C07161=1019.508,345.126,-145.599,171.167,50.075,159.868
C07162=1019.516,345.374,-145.635,171.174,50.072,159.868
C07163=1019.523,345.620,-145.671,171.182,50.070,159.869
C07164=1019.530,345.867,-145.708,171.189,50.068,159.869
C07165=1019.538,346.115,-145.744,171.196,50.066,159.870
C07166=1019.545,346.362,-145.781,171.203,50.064,159.871
C07167=1019.553,346.609,-145.818,171.210,50.062,159.872
C07168=1019.560,346.857,-145.854,171.217,50.060,159.872
C07169=1019.568,347.104,-145.891,171.225,50.058,159.873
C07170=1019.575,347.352,-145.928,171.232,50.055,159.874
C07171=1019.582,347.598,-145.965,171.239,50.054,159.874
C07172=1019.590,347.845,-146.002,171.247,50.052,159.875
C07173=1019.597,348.093,-146.039,171.254,50.050,159.876
C07174=1019.605,348.339,-146.076,171.261,50.048,159.877
C07175=1019.612,348.586,-146.113,171.269,50.046,159.877
C07176=1019.620,348.834,-146.150,171.277,50.044,159.878
C07177=1019.627,349.081,-146.187,171.284,50.042,159.879
C07178=1019.635,349.328,-146.224,171.291,50.040,159.880
C07179=1019.642,349.575,-146.262,171.299,50.038,159.880
C07180=1019.649,349.823,-146.298,171.306,50.036,159.881
C07181=1019.657,350.070,-146.335,171.314,50.034,159.882
C07182=1019.664,350.317,-146.373,171.321,50.033,159.883
C07183=1019.672,350.564,-146.410,171.328,50.031,159.884
C07184=1019.680,350.811,-146.447,171.336,50.029,159.884
C07185=1019.687,351.058,-146.485,171.343,50.027,159.885
C07186=1019.695,351.305,-146.522,171.351,50.025,159.886
C07187=1019.703,351.552,-146.560,171.358,50.023,159.887
C07188=1019.710,351.799,-146.596,171.366,50.021,159.887
C07189=1019.717,352.046,-146.634,171.374,50.020,159.888
C07190=1019.725,352.293,-146.671,171.381,50.018,159.889
C07191=1019.733,352.539,-146.709,171.388,50.016,159.890
C07192=1019.741,352.786,-146.746,171.396,50.015,159.891
C07193=1019.748,353.033,-146.783,171.404,50.013,159.892
C07194=1019.756,353.280,-146.820,171.412,50.011,159.892
C07195=1019.764,353.526,-146.859,171.419,50.009,159.893
C07196=1019.772,353.773,-146.896,171.426,50.007,159.894
C07197=1019.779,354.020,-146.933,171.434,50.005,159.895
C07198=1019.787,354.268,-146.971,171.443,50.004,159.896
C07199=1019.795,354.514,-147.009,171.450,50.002,159.897
C07200=1019.802,354.761,-147.046,171.457,50.000,159.897
C07201=1019.810,355.008,-147.084,171.465,49.999,159.898
C07202=1019.818,355.256,-147.122,171.473,49.998,159.899
C07203=1019.825,355.503,-147.160,171.480,49.996,159.900
C07204=1019.833,355.749,-147.197,171.489,49.994,159.901
C07205=1019.841,355.997,-147.235,171.496,49.993,159.902
C07206=1019.848,356.244,-147.274,171.503,49.991,159.903
C07207=1019.856,356.491,-147.311,171.511,49.990,159.904
C07208=1019.864,356.738,-147.350,171.520,49.987,159.905
C07209=1019.872,356.984,-147.387,171.527,49.986,159.906
C07210=1019.880,357.232,-147.425,171.535,49.985,159.906
C07211=1019.888,357.478,-147.463,171.543,49.983,159.907
C07212=1019.895,357.726,-147.501,171.551,49.981,159.908
C07213=1019.903,357.973,-147.540,171.559,49.980,159.909
C07214=1019.910,358.219,-147.578,171.567,49.979,159.910
C07215=1019.919,358.466,-147.616,171.575,49.977,159.911
C07216=1019.927,358.713,-147.653,171.583,49.976,159.912
C07217=1019.935,358.961,-147.692,171.590,49.975,159.913
C07218=1019.942,359.207,-147.730,171.598,49.973,159.914
C07219=1019.950,359.454,-147.769,171.607,49.971,159.915
C07220=1019.958,359.701,-147.807,171.614,49.970,159.916
C07221=1019.966,359.948,-147.846,171.622,49.969,159.917
C07222=1019.974,360.195,-147.884,171.631,49.967,159.918
C07223=1019.982,360.442,-147.923,171.638,49.966,159.919
C07224=1019.989,360.688,-147.961,171.646,49.965,159.920
C07225=1019.997,360.936,-148.000,171.655,49.963,159.921
C07226=1020.005,361.183,-148.039,171.663,49.962,159.922
C07227=1020.013,361.430,-148.077,171.670,49.961,159.923
C07228=1020.021,361.676,-148.116,171.678,49.960,159.924
C07229=1020.029,361.923,-148.154,171.687,49.958,159.925
C07230=1020.037,362.170,-148.193,171.695,49.957,159.926
C07231=1020.045,362.417,-148.232,171.703,49.955,159.927
C07232=1020.053,362.663,-148.271,171.711,49.954,159.928
C07233=1020.060,362.910,-148.310,171.719,49.953,159.929
C07234=1020.068,363.158,-148.348,171.728,49.952,159.930
C07235=1020.077,363.404,-148.388,171.735,49.951,159.931
C07236=1020.084,363.651,-148.426,171.743,49.949,159.932
C07237=1020.092,363.898,-148.465,171.752,49.948,159.933
C07238=1020.101,364.145,-148.504,171.760,49.947,159.934
C07239=1020.109,364.392,-148.543,171.769,49.946,159.935
C07240=1020.117,364.638,-148.581,171.777,49.945,159.936
C07241=1020.124,364.885,-148.621,171.785,49.943,159.937
C07242=1020.133,365.132,-148.660,171.794,49.943,159.939
C07243=1020.141,365.379,-148.699,171.802,49.941,159.940
C07244=1020.149,365.626,-148.738,171.810,49.940,159.941
C07245=1020.158,365.872,-148.777,171.818,49.939,159.942
C07246=1020.166,366.119,-148.816,171.827,49.938,159.943
C07247=1020.174,366.366,-148.855,171.835,49.937,159.944
C07248=1020.182,366.620,-148.895,171.844,49.936,159.945
C07249=1020.191,366.874,-148.936,171.853,49.934,159.946
C07250=1020.199,367.127,-148.977,171.862,49.933,159.947
C07251=1020.208,367.381,-149.017,171.870,49.932,159.948
C07252=1020.216,367.628,-149.056,171.879,49.931,159.950
C07253=1020.225,367.875,-149.095,171.887,49.930,159.951
C07254=1020.232,368.122,-149.135,171.896,49.929,159.952
C07255=1020.241,368.369,-149.174,171.904,49.929,159.953
C07256=1020.249,368.615,-149.213,171.913,49.927,159.954
C07257=1020.257,368.861,-149.254,171.922,49.926,159.956
C07258=1020.266,369.108,-149.293,171.930,49.926,159.957
C07259=1020.273,369.355,-149.333,171.939,49.925,159.958
C07260=1020.282,369.602,-149.373,171.947,49.924,159.959
C07261=1020.290,369.848,-149.413,171.956,49.923,159.960
C07262=1020.298,370.095,-149.452,171.964,49.922,159.961
C07263=1020.306,370.341,-149.493,171.973,49.921,159.963
C07264=1020.315,370.588,-149.532,171.981,49.921,159.964
C07265=1020.322,370.835,-149.572,171.990,49.920,159.965
C07266=1020.332,371.082,-149.612,171.999,49.918,159.966
C07267=1020.339,371.328,-149.652,172.007,49.918,159.967
C07268=1020.348,371.575,-149.691,172.017,49.917,159.969
C07269=1020.356,371.821,-149.732,172.026,49.916,159.970
C07270=1020.364,372.068,-149.771,172.034,49.916,159.971
C07271=1020.374,372.315,-149.812,172.043,49.915,159.973
C07272=1020.381,372.562,-149.852,172.052,49.914,159.974
C07273=1020.390,372.807,-149.892,172.060,49.913,159.975
C07274=1020.398,373.054,-149.932,172.070,49.913,159.976
C07275=1020.407,373.301,-149.972,172.079,49.912,159.978
C07276=1020.415,373.548,-150.012,172.087,49.911,159.979
C07277=1020.424,373.794,-150.052,172.096,49.911,159.980
C07278=1020.432,374.041,-150.093,172.105,49.910,159.981
C07279=1020.441,374.288,-150.132,172.113,49.909,159.983
C07280=1020.449,374.535,-150.173,172.123,49.909,159.984
C07281=1020.458,374.780,-150.213,172.132,49.908,159.985
C07282=1020.466,375.027,-150.254,172.141,49.907,159.987
C07283=1020.475,375.274,-150.294,172.150,49.907,159.988
C07284=1020.483,375.520,-150.334,172.159,49.906,159.989
C07285=1020.493,375.767,-150.375,172.168,49.905,159.991
C07286=1020.501,376.013,-150.415,172.178,49.905,159.992
C07287=1020.510,376.260,-150.456,172.187,49.904,159.993
C07288=1020.518,376.506,-150.496,172.195,49.904,159.995
C07289=1020.527,376.753,-150.537,172.204,49.903,159.996
C07290=1020.535,377.000,-150.578,172.214,49.903,159.998
C07291=1020.544,377.246,-150.619,172.223,49.902,159.999
C07292=1020.552,377.492,-150.660,172.232,49.902,160.000
C07293=1020.561,377.739,-150.701,172.241,49.902,160.002
C07294=1020.569,377.985,-150.741,172.250,49.901,160.003
C07295=1020.578,378.232,-150.782,172.260,49.900,160.005
C07296=1020.587,378.478,-150.824,172.269,49.900,160.006
C07297=1020.595,378.724,-150.864,172.279,49.900,160.007
C07298=1020.604,378.971,-150.906,172.288,49.899,160.009
C07299=1020.613,379.218,-150.947,172.297,49.899,160.010
C07300=1020.621,379.464,-150.988,172.306,49.899,160.012
C07301=1020.630,379.710,-151.029,172.315,49.898,160.013
C07302=1020.639,379.957,-151.070,172.325,49.898,160.015
C07303=1020.648,380.203,-151.111,172.334,49.898,160.016
C07304=1020.657,380.449,-151.153,172.344,49.897,160.018
C07305=1020.665,380.696,-151.194,172.353,49.897,160.019
C07306=1020.674,380.943,-151.236,172.363,49.897,160.021
C07307=1020.683,381.190,-151.277,172.372,49.896,160.022
C07308=1020.693,381.465,-151.322,172.383,49.896,160.024
C07309=1020.703,381.741,-151.368,172.394,49.896,160.025
C07310=1020.712,382.017,-151.415,172.405,49.896,160.027
C07311=1020.723,382.292,-151.462,172.415,49.895,160.029
C07312=1020.731,382.539,-151.503,172.425,49.895,160.030
C07313=1020.740,382.786,-151.545,172.435,49.895,160.032
C07314=1020.750,383.032,-151.586,172.444,49.895,160.033
C07315=1020.759,383.278,-151.628,172.454,49.894,160.035
C07316=1020.768,383.525,-151.669,172.463,49.894,160.036
C07317=1020.777,383.771,-151.711,172.473,49.894,160.038
C07318=1020.786,384.017,-151.753,172.483,49.894,160.040
C07319=1020.795,384.263,-151.794,172.492,49.893,160.041
C07320=1020.804,384.510,-151.836,172.503,49.893,160.043
C07321=1020.813,384.756,-151.877,172.513,49.893,160.044
C07322=1020.822,385.002,-151.919,172.522,49.893,160.046
C07323=1020.831,385.249,-151.961,172.532,49.893,160.047
C07324=1020.840,385.495,-152.003,172.542,49.893,160.049
C07325=1020.849,385.741,-152.045,172.551,49.893,160.051
C07326=1020.859,385.988,-152.087,172.562,49.893,160.052
C07327=1020.868,386.234,-152.129,172.572,49.893,160.054
C07328=1020.877,386.480,-152.171,172.582,49.893,160.056
C07329=1020.886,386.726,-152.214,172.592,49.893,160.057
C07330=1020.895,386.972,-152.255,172.601,49.893,160.059
C07331=1020.904,387.218,-152.298,172.612,49.893,160.060
C07332=1020.914,387.465,-152.340,172.622,49.893,160.062
C07333=1020.923,387.711,-152.382,172.632,49.893,160.064
C07334=1020.932,387.957,-152.424,172.642,49.893,160.066
C07335=1020.941,388.203,-152.466,172.652,49.893,160.067
C07336=1020.951,388.449,-152.509,172.662,49.894,160.069
C07337=1020.959,388.696,-152.551,172.672,49.894,160.071
C07338=1020.969,388.942,-152.594,172.682,49.894,160.072
C07339=1020.978,389.188,-152.637,172.693,49.894,160.074
C07340=1020.988,389.434,-152.679,172.703,49.894,160.076
C07341=1020.996,389.680,-152.722,172.713,49.894,160.078
C07342=1021.006,389.926,-152.765,172.724,49.894,160.079
C07343=1021.015,390.172,-152.807,172.734,49.895,160.081
C07344=1021.025,390.419,-152.850,172.744,49.895,160.083
C07345=1021.034,390.664,-152.893,172.754,49.895,160.084
C07346=1021.043,390.911,-152.936,172.765,49.896,160.086
C07347=1021.053,391.157,-152.978,172.776,49.895,160.088
C07348=1021.063,391.403,-153.021,172.785,49.896,160.090
C07349=1021.072,391.648,-153.064,172.796,49.897,160.092
C07350=1021.081,391.895,-153.108,172.807,49.896,160.094
C07351=1021.090,392.141,-153.150,172.816,49.897,160.095
C07352=1021.100,392.387,-153.193,172.828,49.897,160.097
C07353=1021.110,392.632,-153.236,172.838,49.897,160.099
C07354=1021.119,392.879,-153.280,172.849,49.898,160.101
C07355=1021.129,393.126,-153.322,172.859,49.898,160.103
C07356=1021.138,393.371,-153.366,172.870,49.899,160.105
C07357=1021.147,393.618,-153.409,172.880,49.899,160.106
C07358=1021.158,393.863,-153.452,172.891,49.899,160.108
C07359=1021.166,394.109,-153.496,172.902,49.900,160.110
C07360=1021.176,394.355,-153.539,172.913,49.901,160.112
C07361=1021.186,394.601,-153.583,172.923,49.901,160.114
C07362=1021.195,394.846,-153.626,172.934,49.901,160.116
C07363=1021.205,395.093,-153.669,172.945,49.902,160.118
C07364=1021.214,395.339,-153.713,172.955,49.903,160.120
C07365=1021.225,395.585,-153.757,172.967,49.903,160.122
C07366=1021.234,395.831,-153.801,172.977,49.904,160.124
C07367=1021.244,396.076,-153.844,172.988,49.904,160.125
C07368=1021.256,396.390,-153.900,173.002,49.905,160.128
C07369=1021.268,396.703,-153.955,173.016,49.906,160.131
C07370=1021.281,397.017,-154.011,173.030,49.906,160.133
C07371=1021.294,397.330,-154.066,173.044,49.907,160.135
C07372=1021.303,397.576,-154.110,173.055,49.907,160.137
C07373=1021.313,397.822,-154.155,173.067,49.908,160.140
C07374=1021.323,398.067,-154.199,173.078,49.909,160.142
C07375=1021.333,398.313,-154.243,173.088,49.910,160.143
C07376=1021.343,398.559,-154.286,173.099,49.910,160.145
C07377=1021.352,398.805,-154.331,173.111,49.911,160.148
C07378=1021.363,399.051,-154.375,173.122,49.912,160.150
C07379=1021.372,399.297,-154.419,173.134,49.913,160.152
C07380=1021.382,399.542,-154.464,173.144,49.913,160.154
C07381=1021.392,399.788,-154.507,173.155,49.914,160.156
C07382=1021.402,400.034,-154.552,173.167,49.915,160.158
C07383=1021.412,400.280,-154.597,173.179,49.916,160.160
C07384=1021.422,400.526,-154.641,173.190,49.916,160.162
C07385=1021.432,400.771,-154.686,173.202,49.917,160.164
C07386=1021.441,401.017,-154.730,173.213,49.918,160.166
C07387=1021.452,401.263,-154.774,173.225,49.919,160.169
C07388=1021.462,401.509,-154.819,173.236,49.920,160.171
C07389=1021.472,401.754,-154.864,173.248,49.921,160.173
C07390=1021.481,402.000,-154.909,173.259,49.922,160.175
C07391=1021.492,402.246,-154.954,173.271,49.922,160.177
C07392=1021.501,402.491,-154.999,173.282,49.923,160.179
C07393=1021.512,402.737,-155.043,173.294,49.924,160.181
C07394=1021.522,402.983,-155.088,173.306,49.925,160.184
C07395=1021.532,403.228,-155.133,173.317,49.926,160.186
C07396=1021.542,403.475,-155.178,173.329,49.927,160.188
C07397=1021.552,403.720,-155.223,173.341,49.928,160.190
C07398=1021.563,403.965,-155.268,173.352,49.929,160.192
C07399=1021.573,404.211,-155.313,173.364,49.931,160.195
C07400=1021.583,404.456,-155.358,173.376,49.932,160.197
C07401=1021.593,404.702,-155.404,173.388,49.933,160.199
C07402=1021.604,404.948,-155.449,173.399,49.934,160.202
C07403=1021.613,405.194,-155.494,173.412,49.935,160.204
C07404=1021.625,405.439,-155.539,173.424,49.936,160.206
C07405=1021.634,405.684,-155.584,173.436,49.937,160.208
C07406=1021.645,405.930,-155.630,173.448,49.939,160.211
C07407=1021.655,406.176,-155.675,173.460,49.939,160.213
C07408=1021.666,406.422,-155.721,173.472,49.941,160.216
C07409=1021.677,406.666,-155.766,173.484,49.942,160.218
C07410=1021.687,406.913,-155.811,173.496,49.943,160.220
C07411=1021.698,407.158,-155.857,173.509,49.944,160.222
C07412=1021.708,407.404,-155.903,173.521,49.945,160.225
C07413=1021.719,407.650,-155.948,173.533,49.946,160.227
C07414=1021.729,407.895,-155.994,173.545,49.948,160.230
C07415=1021.740,408.140,-156.039,173.557,49.949,160.232
C07416=1021.751,408.386,-156.085,173.570,49.950,160.234
C07417=1021.761,408.631,-156.131,173.582,49.951,160.237
C07418=1021.772,408.877,-156.177,173.595,49.952,160.239
C07419=1021.782,409.123,-156.223,173.607,49.954,160.242
C07420=1021.793,409.368,-156.269,173.620,49.955,160.244
C07421=1021.804,409.614,-156.314,173.632,49.957,160.246
C07422=1021.815,409.859,-156.361,173.645,49.958,160.249
C07423=1021.825,410.104,-156.407,173.657,49.959,160.251
C07424=1021.836,410.350,-156.453,173.671,49.961,160.254
C07425=1021.846,410.595,-156.500,173.683,49.963,160.256
C07426=1021.857,410.841,-156.546,173.696,49.964,160.259
C07427=1021.868,411.086,-156.593,173.708,49.965,160.261
C07428=1021.881,411.399,-156.652,173.724,49.968,160.265
C07429=1021.895,411.712,-156.711,173.741,49.969,160.268
C07430=1021.910,412.026,-156.770,173.757,49.971,160.271
C07431=1021.923,412.338,-156.829,173.773,49.973,160.274
C07432=1021.934,412.584,-156.876,173.786,49.975,160.277
C07433=1021.945,412.829,-156.923,173.799,49.976,160.280
C07434=1021.956,413.074,-156.969,173.813,49.978,160.282
C07435=1021.967,413.320,-157.016,173.825,49.979,160.285
C07436=1021.978,413.565,-157.063,173.838,49.981,160.287
C07437=1021.989,413.810,-157.110,173.852,49.983,160.290
C07438=1022.000,414.055,-157.157,173.865,49.984,160.293
C07439=1022.011,414.300,-157.203,173.878,49.986,160.295
C07440=1022.022,414.546,-157.251,173.892,49.987,160.298
C07441=1022.033,414.791,-157.298,173.904,49.989,160.301
C07442=1022.045,415.037,-157.345,173.917,49.991,160.303
C07443=1022.056,415.283,-157.392,173.931,49.993,160.306
C07444=1022.067,415.528,-157.438,173.944,49.994,160.309
C07445=1022.078,415.773,-157.486,173.958,49.996,160.312
C07446=1022.089,416.018,-157.533,173.971,49.998,160.314
C07447=1022.100,416.263,-157.581,173.985,49.999,160.317
C07448=1022.112,416.509,-157.628,173.998,50.002,160.320
C07449=1022.122,416.754,-157.676,174.012,50.003,160.323
C07450=1022.134,416.999,-157.723,174.025,50.005,160.325
C07451=1022.146,417.244,-157.771,174.039,50.007,160.328
C07452=1022.156,417.489,-157.819,174.052,50.009,160.331
C07453=1022.168,417.735,-157.866,174.067,50.011,160.334
C07454=1022.179,417.980,-157.914,174.081,50.013,160.337
C07455=1022.191,418.225,-157.962,174.094,50.015,160.340
C07456=1022.202,418.470,-158.010,174.108,50.016,160.342
C07457=1022.213,418.716,-158.058,174.122,50.019,160.345
C07458=1022.225,418.960,-158.105,174.136,50.021,160.348
C07459=1022.236,419.205,-158.154,174.150,50.022,160.351
C07460=1022.248,419.450,-158.201,174.164,50.024,160.354
C07461=1022.259,419.695,-158.249,174.177,50.027,160.357
C07462=1022.271,419.941,-158.297,174.192,50.028,160.360
C07463=1022.282,420.186,-158.345,174.206,50.031,160.363
C07464=1022.294,420.432,-158.394,174.221,50.033,160.366
C07465=1022.306,420.676,-158.442,174.235,50.035,160.369
C07466=1022.318,420.921,-158.490,174.249,50.037,160.372
C07467=1022.329,421.167,-158.538,174.263,50.039,160.375
C07468=1022.341,421.411,-158.586,174.277,50.041,160.378
C07469=1022.352,421.657,-158.635,174.292,50.043,160.381
C07470=1022.365,421.902,-158.684,174.306,50.045,160.384
C07471=1022.376,422.147,-158.732,174.321,50.047,160.387
C07472=1022.389,422.415,-158.785,174.336,50.050,160.390
C07473=1022.402,422.683,-158.839,174.352,50.052,160.393
C07474=1022.415,422.951,-158.892,174.369,50.054,160.397
C07475=1022.428,423.219,-158.945,174.384,50.057,160.400
C07476=1022.439,423.463,-158.994,174.399,50.059,160.403
C07477=1022.451,423.709,-159.043,174.414,50.062,160.407
C07478=1022.464,423.953,-159.092,174.428,50.064,160.410
C07479=1022.476,424.199,-159.141,174.443,50.066,160.413
C07480=1022.488,424.443,-159.190,174.459,50.068,160.416
C07481=1022.500,424.689,-159.239,174.474,50.071,160.419
C07482=1022.511,424.933,-159.288,174.488,50.073,160.422
C07483=1022.524,425.178,-159.338,174.503,50.076,160.426
C07484=1022.536,425.423,-159.387,174.518,50.078,160.429
C07485=1022.548,425.668,-159.436,174.534,50.080,160.432
C07486=1022.560,425.913,-159.486,174.549,50.083,160.435
C07487=1022.572,426.157,-159.534,174.564,50.085,160.439
C07488=1022.588,426.479,-159.600,174.584,50.089,160.443
C07489=1022.604,426.800,-159.665,174.604,50.091,160.447
C07490=1022.620,427.120,-159.731,174.624,50.095,160.452
C07491=1022.636,427.441,-159.796,174.644,50.098,160.456
C07492=1022.648,427.685,-159.845,174.660,50.101,160.459
C07493=1022.661,427.930,-159.895,174.675,50.103,160.463
C07494=1022.673,428.175,-159.945,174.691,50.106,160.466
C07495=1022.685,428.420,-159.996,174.706,50.109,160.470
C07496=1022.697,428.665,-160.046,174.722,50.111,160.473
C07497=1022.710,428.909,-160.096,174.738,50.114,160.476
C07498=1022.723,429.154,-160.145,174.754,50.116,160.480
C07499=1022.735,429.399,-160.195,174.769,50.119,160.483
C07500=1022.747,429.643,-160.245,174.785,50.122,160.487
C07501=1022.760,429.888,-160.296,174.802,50.125,160.490
C07502=1022.772,430.133,-160.346,174.817,50.127,160.494
C07503=1022.785,430.377,-160.396,174.834,50.130,160.497
C07504=1022.799,430.622,-160.447,174.849,50.133,160.501
C07505=1022.811,430.867,-160.497,174.866,50.135,160.504
C07506=1022.824,431.111,-160.548,174.881,50.138,160.508
C07507=1022.836,431.355,-160.599,174.898,50.141,160.511
C07508=1022.849,431.601,-160.649,174.914,50.144,160.515
C07509=1022.862,431.845,-160.700,174.931,50.147,160.519
C07510=1022.875,432.089,-160.750,174.947,50.149,160.522
C07511=1022.888,432.334,-160.801,174.964,50.152,160.526
C07512=1022.901,432.578,-160.851,174.980,50.155,160.529
C07513=1022.914,432.823,-160.903,174.997,50.158,160.533
C07514=1022.927,433.067,-160.954,175.013,50.161,160.537
C07515=1022.939,433.311,-161.005,175.030,50.164,160.540
C07516=1022.953,433.556,-161.056,175.047,50.166,160.544
C07517=1022.965,433.800,-161.107,175.064,50.169,160.548
C07518=1022.978,434.045,-161.158,175.081,50.172,160.552
C07519=1022.992,434.289,-161.210,175.097,50.176,160.555
C07520=1023.005,434.534,-161.261,175.114,50.179,160.559
C07521=1023.018,434.778,-161.313,175.131,50.182,160.563
C07522=1023.031,435.023,-161.365,175.148,50.185,160.567
C07523=1023.044,435.267,-161.416,175.165,50.188,160.571
C07524=1023.057,435.512,-161.467,175.182,50.191,160.574
C07525=1023.070,435.756,-161.519,175.199,50.194,160.578
C07526=1023.084,436.000,-161.571,175.217,50.197,160.582
C07527=1023.097,436.244,-161.623,175.235,50.200,160.586
C07528=1023.110,436.488,-161.674,175.252,50.203,160.590
C07529=1023.124,436.732,-161.726,175.269,50.207,160.594
C07530=1023.137,436.977,-161.778,175.286,50.210,160.598
C07531=1023.150,437.221,-161.831,175.304,50.212,160.602
C07532=1023.164,437.465,-161.883,175.322,50.216,160.606
C07533=1023.177,437.710,-161.934,175.339,50.219,160.610
C07534=1023.191,437.954,-161.986,175.357,50.222,160.614
C07535=1023.204,438.198,-162.039,175.375,50.226,160.618
C07536=1022.814,436.266,-161.961,175.226,50.266,160.605
C07537=1022.801,436.022,-161.909,175.209,50.264,160.601
C07538=1022.788,435.777,-161.858,175.191,50.260,160.597
C07539=1022.774,435.533,-161.806,175.174,50.257,160.593
C07540=1022.761,435.289,-161.754,175.157,50.254,160.589
C07541=1022.748,435.044,-161.703,175.139,50.252,160.585
C07542=1022.735,434.800,-161.651,175.122,50.248,160.581
C07543=1022.722,434.556,-161.600,175.105,50.245,160.578
C07544=1022.708,434.312,-161.549,175.088,50.243,160.574
C07545=1022.695,434.067,-161.497,175.071,50.240,160.570
C07546=1022.683,433.823,-161.447,175.054,50.237,160.567
C07547=1022.669,433.578,-161.395,175.038,50.234,160.563
C07548=1022.656,433.334,-161.344,175.021,50.231,160.559
C07549=1022.643,433.089,-161.293,175.004,50.228,160.555
C07550=1022.631,432.845,-161.242,174.988,50.226,160.552
C07551=1022.618,432.601,-161.191,174.971,50.223,160.548
C07552=1022.605,432.356,-161.140,174.955,50.220,160.544
C07553=1022.592,432.112,-161.089,174.938,50.217,160.541
C07554=1022.579,431.867,-161.038,174.922,50.215,160.537
C07555=1022.567,431.622,-160.988,174.905,50.212,160.534
C07556=1022.554,431.378,-160.937,174.889,50.209,160.530
C07557=1022.540,431.133,-160.886,174.873,50.206,160.526
C07558=1022.528,430.888,-160.836,174.857,50.204,160.523
C07559=1022.515,430.644,-160.786,174.840,50.201,160.519
C07560=1022.503,430.399,-160.735,174.825,50.198,160.516
C07561=1022.490,430.154,-160.685,174.808,50.196,160.512
C07562=1022.477,429.911,-160.635,174.792,50.193,160.509
C07563=1022.464,429.665,-160.585,174.776,50.191,160.505
C07564=1022.452,429.420,-160.535,174.760,50.188,160.502
C07565=1022.439,429.176,-160.484,174.744,50.186,160.499
C07566=1022.427,428.931,-160.434,174.729,50.183,160.495
C07567=1022.415,428.686,-160.384,174.713,50.180,160.492
C07568=1022.402,428.442,-160.334,174.697,50.178,160.488
C07569=1022.390,428.198,-160.284,174.681,50.176,160.485
C07570=1022.378,427.953,-160.234,174.666,50.173,160.482
C07571=1022.365,427.708,-160.184,174.650,50.170,160.478
C07572=1022.353,427.463,-160.135,174.635,50.168,160.475
C07573=1022.338,427.163,-160.074,174.616,50.165,160.471
C07574=1022.323,426.862,-160.012,174.596,50.162,160.467
C07575=1022.308,426.561,-159.952,174.578,50.159,160.463
C07576=1022.294,426.261,-159.890,174.559,50.156,160.458
C07577=1022.281,426.016,-159.841,174.543,50.154,160.455
C07578=1022.269,425.771,-159.792,174.528,50.152,160.452
C07579=1022.257,425.526,-159.742,174.513,50.149,160.449
C07580=1022.245,425.281,-159.692,174.498,50.147,160.445
C07581=1022.233,425.037,-159.644,174.483,50.145,160.442
C07582=1022.221,424.791,-159.594,174.468,50.143,160.439
C07583=1022.209,424.546,-159.545,174.454,50.140,160.436
C07584=1022.197,424.301,-159.497,174.438,50.138,160.433
C07585=1022.185,424.057,-159.448,174.424,50.136,160.430
C07586=1022.172,423.811,-159.399,174.408,50.134,160.426
C07587=1022.161,423.567,-159.350,174.394,50.132,160.423
C07588=1022.149,423.321,-159.300,174.379,50.129,160.420
C07589=1022.137,423.077,-159.252,174.364,50.127,160.417
C07590=1022.125,422.832,-159.203,174.349,50.125,160.414
C07591=1022.113,422.587,-159.154,174.335,50.123,160.411
C07592=1022.102,422.342,-159.106,174.321,50.121,160.408
C07593=1022.090,422.097,-159.057,174.305,50.119,160.405
C07594=1022.078,421.852,-159.008,174.292,50.116,160.402
C07595=1022.067,421.607,-158.960,174.277,50.115,160.399
C07596=1022.055,421.362,-158.911,174.263,50.112,160.396
C07597=1022.043,421.116,-158.863,174.248,50.111,160.393
C07598=1022.031,420.872,-158.815,174.234,50.108,160.390
C07599=1022.020,420.627,-158.766,174.220,50.107,160.387
C07600=1022.008,420.382,-158.719,174.206,50.104,160.384
C07601=1021.996,420.137,-158.671,174.191,50.103,160.381
C07602=1021.985,419.891,-158.623,174.177,50.100,160.378
C07603=1021.973,419.647,-158.574,174.163,50.099,160.375
C07604=1021.962,419.401,-158.526,174.149,50.097,160.372
C07605=1021.950,419.156,-158.478,174.135,50.095,160.369
C07606=1021.938,418.911,-158.430,174.121,50.093,160.366
C07607=1021.927,418.666,-158.382,174.107,50.091,160.364
C07608=1021.916,418.420,-158.335,174.093,50.090,160.361
C07609=1021.904,418.175,-158.287,174.078,50.088,160.358
C07610=1021.893,417.930,-158.239,174.065,50.086,160.355
C07611=1021.881,417.685,-158.192,174.051,50.084,160.352
C07612=1021.870,417.440,-158.144,174.038,50.082,160.349
C07613=1021.859,417.194,-158.097,174.024,50.081,160.347
C07614=1021.848,416.949,-158.048,174.010,50.079,160.344
C07615=1021.837,416.704,-158.002,173.996,50.077,160.341
C07616=1021.825,416.459,-157.954,173.983,50.075,160.338
C07617=1021.814,416.213,-157.906,173.969,50.074,160.335
C07618=1021.803,415.969,-157.859,173.956,50.072,160.333
C07619=1021.792,415.723,-157.811,173.942,50.070,160.330
C07620=1021.780,415.478,-157.764,173.929,50.069,160.327
C07621=1021.764,415.118,-157.695,173.909,50.066,160.323
C07622=1021.748,414.757,-157.625,173.890,50.064,160.319
C07623=1021.731,414.397,-157.557,173.870,50.062,160.315
C07624=1021.715,414.036,-157.488,173.851,50.059,160.311
C07625=1021.704,413.791,-157.441,173.838,50.057,160.309
C07626=1021.693,413.546,-157.394,173.825,50.056,160.306
C07627=1021.682,413.301,-157.348,173.811,50.054,160.304
C07628=1021.671,413.056,-157.301,173.798,50.053,160.301
C07629=1021.660,412.821,-157.256,173.786,50.051,160.298
C07630=1021.650,412.587,-157.212,173.773,50.050,160.296
C07631=1021.639,412.352,-157.167,173.761,50.049,160.293
C07632=1021.629,412.118,-157.122,173.749,50.047,160.291
C07633=1021.619,411.884,-157.078,173.736,50.046,160.289
C07634=1021.608,411.648,-157.034,173.724,50.045,160.286
C07635=1021.598,411.414,-156.990,173.712,50.044,160.284
C07636=1021.588,411.180,-156.945,173.700,50.042,160.281
C07637=1021.578,410.935,-156.899,173.687,50.041,160.279
C07638=1021.567,410.690,-156.853,173.673,50.039,160.276
C07639=1021.555,410.443,-156.806,173.661,50.038,160.274
C07640=1021.545,410.198,-156.760,173.648,50.037,160.271
C07641=1021.534,409.953,-156.714,173.636,50.035,160.269
C07642=1021.524,409.707,-156.667,173.623,50.034,160.266
C07643=1021.513,409.461,-156.621,173.610,50.033,160.264
C07644=1021.502,409.216,-156.575,173.598,50.031,160.261
C07645=1021.492,408.971,-156.529,173.585,50.030,160.259
C07646=1021.481,408.725,-156.483,173.573,50.029,160.257
C07647=1021.471,408.479,-156.438,173.560,50.028,160.254
C07648=1021.460,408.234,-156.392,173.548,50.026,160.252
C07649=1021.449,407.988,-156.347,173.536,50.026,160.250
C07650=1021.438,407.742,-156.301,173.524,50.024,160.247
C07651=1021.428,407.497,-156.255,173.511,50.023,160.245
C07652=1021.418,407.252,-156.209,173.499,50.022,160.242
C07653=1021.407,407.006,-156.164,173.487,50.021,160.240
C07654=1021.396,406.760,-156.119,173.474,50.020,160.238
C07655=1021.385,406.515,-156.073,173.463,50.019,160.235
C07656=1021.376,406.269,-156.028,173.451,50.018,160.233
C07657=1021.365,406.024,-155.982,173.438,50.017,160.231
C07658=1021.355,405.777,-155.937,173.426,50.016,160.229
C07659=1021.344,405.533,-155.892,173.414,50.014,160.226
C07660=1021.334,405.287,-155.847,173.402,50.014,160.224
C07661=1021.323,405.041,-155.801,173.390,50.013,160.222
C07662=1021.313,404.796,-155.756,173.378,50.012,160.219
C07663=1021.303,404.549,-155.711,173.367,50.011,160.217
C07664=1021.292,404.305,-155.666,173.353,50.010,160.215
C07665=1021.282,404.059,-155.621,173.342,50.009,160.212
C07666=1021.272,403.813,-155.576,173.330,50.008,160.210
C07667=1021.262,403.567,-155.531,173.318,50.007,160.208
C07668=1021.252,403.321,-155.486,173.307,50.006,160.206
C07669=1021.242,403.076,-155.442,173.295,50.005,160.204
C07670=1021.231,402.830,-155.396,173.284,50.004,160.202
C07671=1021.221,402.585,-155.351,173.271,50.004,160.199
C07672=1021.212,402.339,-155.306,173.260,50.003,160.197
C07673=1021.201,402.093,-155.261,173.248,50.002,160.195
C07674=1021.192,401.847,-155.217,173.236,50.001,160.193
C07675=1021.181,401.602,-155.173,173.225,50.000,160.191
C07676=1021.171,401.356,-155.127,173.213,49.999,160.189
C07677=1021.161,401.110,-155.083,173.202,49.998,160.186
C07678=1021.152,400.865,-155.038,173.190,49.998,160.184
C07679=1021.142,400.619,-154.994,173.179,49.997,160.182
C07680=1021.132,400.373,-154.949,173.167,49.996,160.180
C07681=1021.122,400.127,-154.904,173.156,49.995,160.178
C07682=1021.111,399.881,-154.861,173.145,49.995,160.176
C07683=1021.102,399.636,-154.816,173.134,49.994,160.174
C07684=1021.092,399.390,-154.772,173.123,49.993,160.172
C07685=1021.082,399.144,-154.727,173.111,49.993,160.170
C07686=1021.072,398.898,-154.683,173.100,49.992,160.168
C07687=1021.062,398.652,-154.640,173.088,49.991,160.166
C07688=1021.053,398.407,-154.595,173.077,49.991,160.164
C07689=1021.043,398.161,-154.551,173.066,49.991,160.162
C07690=1021.033,397.915,-154.507,173.055,49.990,160.160
C07691=1021.024,397.669,-154.463,173.044,49.989,160.158
C07692=1021.013,397.423,-154.420,173.033,49.988,160.155
C07693=1021.001,397.108,-154.363,173.019,49.988,160.153
C07694=1020.988,396.792,-154.306,173.004,49.987,160.150
C07695=1020.975,396.477,-154.251,172.990,49.986,160.148
C07696=1020.963,396.161,-154.195,172.976,49.986,160.146
C07697=1020.953,395.915,-154.152,172.965,49.986,160.144
C07698=1020.944,395.669,-154.108,172.954,49.985,160.142
C07699=1020.934,395.424,-154.064,172.943,49.984,160.140
C07700=1020.925,395.177,-154.020,172.932,49.985,160.138
C07701=1020.914,394.932,-153.977,172.921,49.984,160.136
C07702=1020.905,394.685,-153.934,172.911,49.983,160.134
C07703=1020.896,394.440,-153.890,172.900,49.983,160.132
C07704=1020.886,394.194,-153.847,172.889,49.983,160.130
C07705=1020.877,393.947,-153.803,172.878,49.982,160.128
C07706=1020.867,393.702,-153.760,172.868,49.982,160.126
C07707=1020.857,393.456,-153.717,172.857,49.981,160.125
C07708=1020.848,393.209,-153.673,172.846,49.982,160.123
C07709=1020.839,392.964,-153.631,172.836,49.981,160.121
C07710=1020.829,392.718,-153.587,172.825,49.981,160.119
C07711=1020.820,392.472,-153.544,172.814,49.981,160.117
C07712=1020.810,392.225,-153.502,172.804,49.980,160.115
C07713=1020.800,391.979,-153.459,172.793,49.980,160.114
C07714=1020.791,391.734,-153.415,172.783,49.980,160.112
C07715=1020.782,391.487,-153.372,172.772,49.980,160.110
C07716=1020.772,391.241,-153.330,172.762,49.979,160.108
C07717=1020.762,390.995,-153.287,172.751,49.980,160.106
C07718=1020.754,390.749,-153.244,172.741,49.979,160.105
C07719=1020.744,390.502,-153.201,172.731,49.979,160.103
C07720=1020.735,390.257,-153.159,172.720,49.979,160.101
C07721=1020.726,390.011,-153.116,172.711,49.979,160.100
C07722=1020.716,389.764,-153.074,172.699,49.978,160.098
C07723=1020.707,389.518,-153.030,172.689,49.978,160.096
C07724=1020.697,389.272,-152.988,172.679,49.978,160.094
C07725=1020.688,389.026,-152.945,172.669,49.979,160.093
C07726=1020.679,388.780,-152.903,172.659,49.978,160.091
C07727=1020.671,388.534,-152.861,172.648,49.979,160.089
C07728=1020.661,388.287,-152.818,172.638,49.978,160.087
C07729=1020.652,388.042,-152.775,172.628,49.978,160.086
C07730=1020.643,387.795,-152.734,172.617,49.978,160.084
C07731=1020.633,387.549,-152.691,172.608,49.979,160.082
C07732=1020.624,387.303,-152.648,172.598,49.978,160.081
C07733=1020.615,387.057,-152.607,172.588,49.978,160.079
C07734=1020.606,386.811,-152.564,172.578,49.979,160.077
C07735=1020.597,386.565,-152.522,172.568,49.979,160.076
C07736=1020.588,386.318,-152.481,172.558,49.978,160.074
C07737=1020.578,386.072,-152.438,172.547,49.979,160.073
C07738=1020.569,385.825,-152.396,172.537,49.979,160.071
C07739=1020.560,385.580,-152.354,172.528,49.979,160.069
C07740=1020.551,385.333,-152.312,172.518,49.979,160.068
C07741=1020.542,385.087,-152.270,172.508,49.979,160.066
C07742=1020.533,384.841,-152.229,172.498,49.980,160.065
C07743=1020.524,384.594,-152.187,172.488,49.980,160.063
C07744=1020.515,384.348,-152.145,172.479,49.980,160.061
C07745=1020.505,384.102,-152.104,172.469,49.980,160.060
C07746=1020.496,383.855,-152.062,172.459,49.980,160.058
C07747=1020.487,383.609,-152.021,172.449,49.981,160.057
C07748=1020.478,383.363,-151.979,172.439,49.981,160.055
C07749=1020.470,383.116,-151.937,172.430,49.981,160.054
C07750=1020.461,382.870,-151.896,172.420,49.982,160.052
C07751=1020.451,382.624,-151.854,172.411,49.982,160.051
C07752=1020.442,382.378,-151.813,172.401,49.982,160.049
C07753=1020.432,382.100,-151.766,172.390,49.983,160.047
C07754=1020.423,381.821,-151.720,172.379,49.983,160.046
C07755=1020.412,381.542,-151.673,172.368,49.984,160.044
C07756=1020.402,381.264,-151.626,172.357,49.984,160.042
C07757=1020.393,381.018,-151.584,172.347,49.984,160.041
C07758=1020.385,380.771,-151.544,172.338,49.984,160.039
C07759=1020.375,380.525,-151.503,172.329,49.985,160.038
C07760=1020.366,380.279,-151.461,172.319,49.986,160.036
C07761=1020.358,380.032,-151.420,172.310,49.986,160.035
C07762=1020.349,379.786,-151.379,172.300,49.986,160.033
C07763=1020.341,379.539,-151.338,172.291,49.987,160.032
C07764=1020.331,379.293,-151.297,172.281,49.988,160.031
C07765=1020.323,379.047,-151.256,172.272,49.988,160.029
C07766=1020.315,378.800,-151.215,172.262,49.988,160.028
C07767=1020.306,378.554,-151.173,172.253,49.989,160.026
C07768=1020.298,378.307,-151.132,172.245,49.989,160.025
C07769=1020.289,378.060,-151.091,172.235,49.989,160.023
C07770=1020.280,377.814,-151.051,172.226,49.990,160.022
C07771=1020.271,377.568,-151.010,172.216,49.991,160.021
C07772=1020.263,377.322,-150.969,172.207,49.991,160.019
C07773=1020.255,377.075,-150.928,172.198,49.992,160.018
C07774=1020.247,376.828,-150.887,172.188,49.992,160.016
C07775=1020.237,376.582,-150.847,172.179,49.993,160.015
C07776=1020.229,376.335,-150.806,172.171,49.994,160.014
C07777=1020.220,376.089,-150.765,172.161,49.994,160.012
C07778=1020.212,375.842,-150.725,172.152,49.995,160.011
C07779=1020.203,375.595,-150.684,172.143,49.995,160.010
C07780=1020.194,375.350,-150.644,172.134,49.996,160.008
C07781=1020.186,375.103,-150.603,172.125,49.997,160.007
C07782=1020.177,374.857,-150.563,172.115,49.998,160.006
C07783=1020.169,374.609,-150.523,172.107,49.999,160.005
C07784=1020.160,374.363,-150.483,172.098,49.999,160.003
C07785=1020.152,374.117,-150.442,172.089,50.000,160.002
C07786=1020.143,373.869,-150.403,172.079,50.001,160.001
C07787=1020.135,373.623,-150.362,172.070,50.002,159.999
C07788=1020.126,373.377,-150.322,172.062,50.002,159.998
C07789=1020.118,373.130,-150.282,172.053,50.003,159.997
C07790=1020.109,372.884,-150.242,172.044,50.004,159.996
C07791=1020.101,372.637,-150.202,172.035,50.005,159.994
C07792=1020.092,372.390,-150.161,172.027,50.006,159.993
C07793=1020.083,372.143,-150.122,172.017,50.007,159.992
C07794=1020.075,371.897,-150.081,172.008,50.007,159.990
C07795=1020.067,371.651,-150.042,172.000,50.008,159.989
C07796=1020.059,371.404,-150.002,171.991,50.009,159.988
C07797=1020.050,371.157,-149.962,171.982,50.010,159.987
C07798=1020.042,370.910,-149.922,171.973,50.011,159.986
C07799=1020.034,370.663,-149.882,171.965,50.012,159.984
C07800=1020.026,370.417,-149.842,171.956,50.013,159.983
C07801=1020.017,370.171,-149.802,171.947,50.014,159.982
C07802=1020.009,369.924,-149.763,171.939,50.015,159.981
C07803=1020.001,369.677,-149.723,171.930,50.016,159.980
C07804=1019.993,369.430,-149.683,171.922,50.016,159.978
C07805=1019.985,369.184,-149.644,171.913,50.018,159.977
C07806=1019.976,368.938,-149.604,171.904,50.019,159.976
C07807=1019.968,368.691,-149.564,171.896,50.019,159.975
C07808=1019.960,368.444,-149.525,171.887,50.021,159.974
C07809=1019.952,368.197,-149.485,171.879,50.021,159.973
C07810=1019.944,367.951,-149.445,171.870,50.023,159.971
C07811=1019.936,367.704,-149.406,171.861,50.024,159.970
C07812=1019.928,367.456,-149.367,171.853,50.025,159.969
C07813=1019.918,367.200,-149.326,171.844,50.026,159.968
C07814=1019.910,366.945,-149.285,171.835,50.028,159.967
C07815=1019.902,366.689,-149.244,171.826,50.029,159.966
C07816=1019.894,366.433,-149.204,171.817,50.030,159.964
C07817=1019.885,366.186,-149.165,171.809,50.031,159.963
C07818=1019.877,365.939,-149.126,171.801,50.033,159.962
C07819=1019.869,365.692,-149.087,171.792,50.033,159.961
C07820=1019.860,365.445,-149.048,171.784,50.035,159.960
C07821=1019.852,365.199,-149.008,171.776,50.036,159.959
C07822=1019.844,364.951,-148.970,171.767,50.037,159.958
C07823=1019.835,364.705,-148.931,171.759,50.039,159.957
C07824=1019.828,364.458,-148.892,171.750,50.039,159.956
C07825=1019.820,364.211,-148.852,171.742,50.041,159.955
C07826=1019.812,363.964,-148.814,171.734,50.042,159.954
C07827=1019.804,363.717,-148.775,171.726,50.043,159.953
C07828=1019.796,363.471,-148.736,171.717,50.045,159.952
C07829=1019.788,363.224,-148.698,171.709,50.046,159.951
C07830=1019.780,362.977,-148.659,171.701,50.048,159.950
C07831=1019.772,362.731,-148.620,171.693,50.049,159.949
C07832=1019.764,362.483,-148.581,171.684,50.050,159.947
C07833=1019.756,362.236,-148.542,171.676,50.051,159.946
C07834=1019.749,361.989,-148.504,171.667,50.053,159.945
C07835=1019.740,361.743,-148.465,171.660,50.054,159.944
C07836=1019.732,361.496,-148.426,171.652,50.056,159.944
C07837=1019.724,361.249,-148.388,171.644,50.057,159.943
C07838=1019.716,361.002,-148.349,171.636,50.059,159.942
C07839=1019.709,360.755,-148.311,171.627,50.060,159.940
C07840=1019.701,360.508,-148.272,171.619,50.061,159.939
C07841=1019.693,360.261,-148.233,171.611,50.062,159.938
C07842=1019.686,360.014,-148.195,171.603,50.064,159.938
C07843=1019.677,359.767,-148.156,171.595,50.066,159.937
C07844=1019.670,359.520,-148.118,171.588,50.067,159.936
C07845=1019.662,359.273,-148.079,171.579,50.069,159.935
C07846=1019.654,359.027,-148.041,171.571,50.070,159.934
C07847=1019.646,358.779,-148.003,171.564,50.072,159.933
C07848=1019.638,358.533,-147.966,171.555,50.073,159.932
C07849=1019.631,358.286,-147.927,171.547,50.075,159.931
C07850=1019.622,358.039,-147.889,171.539,50.077,159.930
C07851=1019.615,357.792,-147.851,171.531,50.078,159.929
C07852=1019.607,357.545,-147.813,171.524,50.080,159.928
C07853=1019.599,357.298,-147.774,171.515,50.082,159.927
C07854=1019.591,357.050,-147.737,171.508,50.083,159.926
C07855=1019.583,356.804,-147.699,171.500,50.085,159.926
C07856=1019.576,356.557,-147.661,171.492,50.086,159.924
C07857=1019.568,356.310,-147.623,171.484,50.088,159.924
C07858=1019.560,356.063,-147.585,171.477,50.090,159.923
C07859=1019.552,355.816,-147.548,171.469,50.091,159.922
C07860=1019.545,355.568,-147.510,171.461,50.093,159.921
C07861=1019.537,355.322,-147.471,171.453,50.095,159.920
C07862=1019.530,355.075,-147.434,171.446,50.097,159.919
C07863=1019.522,354.828,-147.395,171.437,50.098,159.918
C07864=1019.514,354.581,-147.358,171.430,50.100,159.917
C07865=1019.506,354.334,-147.321,171.422,50.102,159.917
C07866=1019.499,354.087,-147.283,171.415,50.104,159.916
C07867=1019.492,353.840,-147.245,171.406,50.106,159.915
C07868=1019.483,353.592,-147.208,171.399,50.107,159.914
C07869=1019.476,353.345,-147.170,171.392,50.109,159.913
C07870=1019.468,353.098,-147.133,171.384,50.111,159.913
C07871=1019.460,352.851,-147.096,171.376,50.113,159.912
C07872=1019.453,352.605,-147.058,171.368,50.115,159.911
C07873=1019.445,352.356,-147.020,171.361,50.117,159.910
C07874=1019.437,352.107,-146.983,171.354,50.118,159.909
C07875=1019.429,351.858,-146.945,171.345,50.121,159.909
C07876=1019.422,351.609,-146.908,171.338,50.122,159.908
C07877=1019.414,351.362,-146.871,171.330,50.124,159.907
C07878=1019.407,351.115,-146.833,171.323,50.126,159.906
C07879=1019.399,350.868,-146.796,171.315,50.128,159.905
C07880=1019.392,350.621,-146.759,171.307,50.130,159.904
C07881=1019.384,350.374,-146.722,171.300,50.132,159.904
C07882=1019.377,350.127,-146.684,171.293,50.134,159.903
C07883=1019.369,349.880,-146.647,171.286,50.136,159.902
C07884=1019.362,349.633,-146.610,171.278,50.138,159.901
C07885=1019.354,349.386,-146.573,171.270,50.140,159.901
C07886=1019.347,349.139,-146.536,171.263,50.142,159.900
C07887=1019.339,348.892,-146.498,171.255,50.144,159.899
C07888=1019.332,348.644,-146.462,171.248,50.146,159.898
C07889=1019.324,348.397,-146.425,171.241,50.148,159.898
C07890=1019.317,348.150,-146.387,171.233,50.150,159.897
C07891=1019.309,347.902,-146.351,171.226,50.152,159.896
C07892=1019.302,347.655,-146.313,171.218,50.154,159.896
C07893=1019.295,347.408,-146.277,171.211,50.156,159.895
C07894=1019.287,347.161,-146.240,171.204,50.159,159.894
C07895=1019.280,346.915,-146.203,171.196,50.160,159.893
C07896=1019.273,346.667,-146.166,171.189,50.163,159.893
C07897=1019.265,346.419,-146.130,171.182,50.165,159.892
C07898=1019.257,346.173,-146.093,171.175,50.167,159.891
C07899=1019.250,345.925,-146.056,171.168,50.169,159.891
C07900=1019.243,345.677,-146.020,171.159,50.171,159.890
C07901=1019.235,345.431,-145.984,171.152,50.174,159.889
C07902=1019.228,345.184,-145.947,171.145,50.176,159.889
C07903=1019.221,344.936,-145.911,171.138,50.178,159.888
C07904=1019.213,344.689,-145.874,171.131,50.181,159.887
C07905=1019.206,344.442,-145.837,171.124,50.183,159.887
C07906=1019.199,344.195,-145.801,171.117,50.185,159.886
C07907=1019.191,343.947,-145.765,171.110,50.187,159.885
C07908=1019.184,343.700,-145.728,171.103,50.190,159.885
C07909=1019.177,343.453,-145.692,171.096,50.192,159.884
C07910=1019.169,343.206,-145.655,171.088,50.194,159.883
C07911=1019.161,342.959,-145.619,171.081,50.196,159.883
C07912=1019.155,342.712,-145.582,171.073,50.199,159.882
C07913=1019.147,342.464,-145.546,171.066,50.201,159.882
C07914=1019.140,342.217,-145.510,171.059,50.204,159.881
C07915=1019.133,341.970,-145.474,171.052,50.206,159.880
C07916=1019.126,341.722,-145.437,171.045,50.209,159.880
C07917=1019.118,341.475,-145.401,171.038,50.211,159.879
C07918=1019.111,341.227,-145.366,171.031,50.213,159.879
C07919=1019.104,340.980,-145.330,171.024,50.216,159.878
C07920=1019.097,340.733,-145.293,171.017,50.218,159.877
C07921=1019.090,340.485,-145.257,171.010,50.221,159.877
C07922=1019.082,340.239,-145.221,171.003,50.223,159.876
C07923=1019.075,339.991,-145.185,170.996,50.225,159.876
C07924=1019.069,339.743,-145.149,170.989,50.228,159.875
C07925=1019.061,339.496,-145.113,170.982,50.230,159.874
C07926=1019.054,339.249,-145.077,170.975,50.233,159.874
C07927=1019.046,339.002,-145.041,170.968,50.235,159.873
C07928=1019.040,338.754,-145.006,170.961,50.237,159.873
C07929=1019.032,338.507,-144.970,170.954,50.240,159.872
C07930=1019.025,338.260,-144.935,170.947,50.243,159.872
C07931=1019.017,338.012,-144.898,170.940,50.245,159.871
C07932=1019.011,337.765,-144.863,170.933,50.248,159.870
C07933=1019.003,337.513,-144.826,170.926,50.251,159.870
C07934=1018.995,337.262,-144.790,170.919,50.253,159.869
C07935=1018.989,337.010,-144.754,170.912,50.256,159.869
C07936=1018.981,336.759,-144.718,170.905,50.259,159.868
C07937=1018.974,336.512,-144.683,170.899,50.261,159.868
C07938=1018.967,336.265,-144.647,170.892,50.264,159.867
C07939=1018.960,336.017,-144.611,170.885,50.267,159.867
C07940=1018.953,335.770,-144.576,170.878,50.269,159.866
C07941=1018.946,335.523,-144.540,170.871,50.272,159.866
C07942=1018.938,335.275,-144.505,170.864,50.274,159.865
C07943=1018.932,335.027,-144.470,170.858,50.277,159.865
C07944=1018.925,334.780,-144.435,170.851,50.280,159.864
C07945=1018.917,334.533,-144.398,170.844,50.283,159.864
C07946=1018.910,334.285,-144.363,170.837,50.285,159.863
C07947=1018.904,334.038,-144.328,170.830,50.288,159.863
C07948=1018.897,333.790,-144.293,170.823,50.291,159.862
C07949=1018.890,333.542,-144.258,170.817,50.294,159.862
C07950=1018.882,333.296,-144.222,170.810,50.297,159.861
C07951=1018.876,333.048,-144.187,170.803,50.299,159.861
C07952=1018.869,332.801,-144.151,170.797,50.302,159.860
C07953=1018.861,332.554,-144.117,170.789,50.305,159.860
C07954=1018.854,332.306,-144.081,170.783,50.308,159.859
C07955=1018.847,332.058,-144.046,170.776,50.311,159.859
C07956=1018.841,331.811,-144.011,170.770,50.314,159.859
C07957=1018.833,331.564,-143.977,170.763,50.317,159.858
C07958=1018.826,331.317,-143.941,170.757,50.319,159.858
C07959=1018.820,331.069,-143.907,170.750,50.322,159.857
C07960=1018.812,330.821,-143.872,170.744,50.325,159.857
C07961=1018.805,330.574,-143.837,170.737,50.328,159.857
C07962=1018.798,330.326,-143.802,170.730,50.331,159.856
C07963=1018.791,330.079,-143.767,170.724,50.334,159.856
C07964=1018.784,329.831,-143.733,170.717,50.337,159.855
C07965=1018.777,329.584,-143.698,170.710,50.340,159.855
C07966=1018.771,329.336,-143.663,170.703,50.343,159.854
C07967=1018.763,329.089,-143.628,170.697,50.346,159.854
C07968=1018.757,328.841,-143.594,170.690,50.349,159.854
C07969=1018.750,328.594,-143.558,170.684,50.352,159.853
C07970=1018.743,328.347,-143.523,170.678,50.355,159.853
C07971=1018.736,328.099,-143.490,170.671,50.358,159.852
C07972=1018.729,327.852,-143.454,170.665,50.361,159.852
C07973=1018.723,327.604,-143.420,170.658,50.364,159.852
C07974=1018.715,327.357,-143.385,170.651,50.367,159.851
C07975=1018.708,327.109,-143.350,170.645,50.371,159.851
C07976=1018.702,326.861,-143.316,170.638,50.374,159.851
C07977=1018.694,326.614,-143.281,170.632,50.377,159.850
C07978=1018.688,326.366,-143.247,170.626,50.379,159.850
C07979=1018.681,326.119,-143.213,170.620,50.383,159.850
C07980=1018.675,325.872,-143.178,170.613,50.386,159.849
C07981=1018.667,325.624,-143.145,170.607,50.389,159.849
C07982=1018.660,325.377,-143.111,170.600,50.392,159.849
C07983=1018.653,325.129,-143.077,170.593,50.395,159.848
C07984=1018.646,324.881,-143.042,170.587,50.399,159.848
C07985=1018.639,324.634,-143.008,170.581,50.402,159.848
C07986=1018.632,324.386,-142.974,170.574,50.406,159.847
C07987=1018.625,324.138,-142.940,170.568,50.409,159.847
C07988=1018.618,323.890,-142.906,170.561,50.412,159.847
C07989=1018.612,323.643,-142.872,170.555,50.416,159.846
C07990=1018.604,323.396,-142.839,170.548,50.419,159.846
C07991=1018.598,323.148,-142.803,170.543,50.422,159.846
C07992=1018.590,322.901,-142.770,170.536,50.425,159.846
C07993=1018.583,322.645,-142.735,170.529,50.429,159.845
C07994=1018.576,322.389,-142.700,170.522,50.432,159.845
C07995=1018.569,322.134,-142.665,170.516,50.436,159.845
C07996=1018.562,321.878,-142.630,170.510,50.440,159.844
C07997=1018.555,321.631,-142.596,170.503,50.443,159.844
C07998=1018.548,321.383,-142.562,170.497,50.447,159.844
C07999=1018.542,321.136,-142.528,170.490,50.450,159.843
C08000=1018.535,320.887,-142.495,170.485,50.453,159.843
C08001=1018.528,320.640,-142.461,170.479,50.457,159.843
C08002=1018.521,320.392,-142.427,170.472,50.460,159.843
C08003=1018.515,320.145,-142.393,170.466,50.463,159.843
C08004=1018.507,319.897,-142.360,170.460,50.467,159.842
C08005=1018.501,319.650,-142.326,170.453,50.470,159.842
C08006=1018.494,319.402,-142.293,170.447,50.474,159.842
C08007=1018.488,319.154,-142.259,170.442,50.477,159.842
C08008=1018.481,318.907,-142.225,170.435,50.480,159.841
C08009=1018.474,318.659,-142.191,170.429,50.484,159.841
C08010=1018.467,318.411,-142.157,170.422,50.488,159.841
C08011=1018.461,318.164,-142.124,170.416,50.492,159.841
C08012=1018.454,317.916,-142.090,170.409,50.495,159.840
C08013=1018.447,317.669,-142.057,170.404,50.498,159.840
C08014=1018.440,317.421,-142.024,170.398,50.502,159.840
C08015=1018.434,317.173,-141.990,170.392,50.505,159.840
C08016=1018.427,316.926,-141.956,170.386,50.509,159.840
C08017=1018.421,316.678,-141.923,170.379,50.513,159.839
C08018=1018.414,316.430,-141.889,170.373,50.517,159.839
C08019=1018.408,316.182,-141.856,170.367,50.519,159.839
C08020=1018.401,315.935,-141.822,170.361,50.523,159.839
C08021=1018.395,315.687,-141.789,170.355,50.527,159.838
C08022=1018.387,315.439,-141.756,170.349,50.530,159.838
C08023=1018.381,315.192,-141.723,170.342,50.534,159.838
C08024=1018.375,314.945,-141.689,170.337,50.537,159.838
C08025=1018.368,314.696,-141.656,170.331,50.541,159.838
C08026=1018.362,314.449,-141.622,170.325,50.545,159.837
C08027=1018.355,314.201,-141.589,170.318,50.549,159.837
C08028=1018.349,313.954,-141.555,170.312,50.552,159.837
C08029=1018.343,313.706,-141.522,170.307,50.556,159.837
C08030=1018.336,313.459,-141.488,170.301,50.559,159.837
C08031=1018.329,313.211,-141.456,170.294,50.563,159.837
C08032=1018.323,312.963,-141.423,170.289,50.568,159.837
C08033=1018.317,312.715,-141.389,170.282,50.571,159.836
C08034=1018.310,312.468,-141.356,170.277,50.575,159.836
C08035=1018.304,312.220,-141.323,170.271,50.578,159.836
C08036=1018.297,311.973,-141.290,170.265,50.582,159.836
C08037=1018.290,311.725,-141.257,170.258,50.586,159.836
C08038=1018.285,311.477,-141.223,170.253,50.589,159.835
C08039=1018.279,311.229,-141.190,170.247,50.594,159.835
C08040=1018.272,310.982,-141.157,170.241,50.597,159.835
C08041=1018.265,310.734,-141.124,170.235,50.601,159.835
C08042=1018.260,310.486,-141.091,170.229,50.604,159.835
C08043=1018.253,310.239,-141.058,170.223,50.608,159.835
C08044=1018.247,309.991,-141.025,170.217,50.613,159.835
C08045=1018.241,309.743,-140.992,170.211,50.616,159.835
C08046=1018.234,309.496,-140.960,170.206,50.620,159.834
C08047=1018.227,309.248,-140.927,170.200,50.624,159.834
C08048=1018.220,309.000,-140.894,170.194,50.628,159.834
C08049=1018.213,308.753,-140.862,170.188,50.632,159.834
C08050=1018.207,308.505,-140.829,170.182,50.637,159.834
C08051=1018.201,308.257,-140.797,170.176,50.640,159.834
C08052=1018.194,308.009,-140.765,170.170,50.645,159.834
C08053=1018.187,307.759,-140.732,170.164,50.648,159.834
C08054=1018.180,307.509,-140.699,170.158,50.653,159.834
C08055=1018.174,307.258,-140.667,170.153,50.657,159.834
C08056=1018.167,307.009,-140.634,170.147,50.661,159.834
C08057=1018.161,306.761,-140.602,170.141,50.665,159.834
C08058=1018.153,306.513,-140.570,170.135,50.669,159.834
C08059=1018.147,306.265,-140.537,170.129,50.673,159.833
C08060=1018.141,306.017,-140.505,170.123,50.677,159.833
C08061=1018.134,305.769,-140.473,170.117,50.682,159.833
C08062=1018.128,305.521,-140.441,170.112,50.686,159.834
C08063=1018.121,305.274,-140.408,170.106,50.690,159.833
C08064=1018.115,305.026,-140.376,170.100,50.694,159.833
C08065=1018.108,304.778,-140.344,170.094,50.698,159.833
C08066=1018.102,304.531,-140.312,170.088,50.703,159.833
C08067=1018.096,304.283,-140.279,170.082,50.707,159.833
C08068=1018.089,304.035,-140.247,170.077,50.711,159.833
C08069=1018.083,303.787,-140.215,170.071,50.715,159.833
C08070=1018.076,303.539,-140.184,170.066,50.719,159.833
C08071=1018.070,303.292,-140.151,170.060,50.724,159.833
C08072=1018.063,303.044,-140.120,170.054,50.728,159.833
C08073=1018.057,302.796,-140.087,170.048,50.732,159.833
C08074=1018.051,302.548,-140.055,170.043,50.736,159.833
C08075=1018.044,302.300,-140.024,170.037,50.740,159.833
C08076=1018.038,302.052,-139.991,170.031,50.745,159.833
C08077=1018.031,301.805,-139.959,170.025,50.749,159.833
C08078=1018.025,301.556,-139.927,170.019,50.754,159.833
C08079=1018.018,301.309,-139.895,170.015,50.758,159.833
C08080=1018.012,301.061,-139.863,170.009,50.762,159.833
C08081=1018.005,300.813,-139.832,170.003,50.766,159.833
C08082=1017.999,300.565,-139.799,169.997,50.771,159.833
C08083=1017.993,300.317,-139.767,169.991,50.775,159.833
C08084=1017.987,300.070,-139.736,169.986,50.779,159.833
C08085=1017.981,299.822,-139.704,169.980,50.784,159.833
C08086=1017.974,299.574,-139.672,169.975,50.788,159.833
C08087=1017.968,299.326,-139.640,169.969,50.792,159.833
C08088=1017.961,299.078,-139.608,169.963,50.797,159.833
C08089=1017.955,298.830,-139.576,169.958,50.801,159.833
C08090=1017.949,298.583,-139.545,169.953,50.806,159.833
C08091=1017.943,298.335,-139.513,169.947,50.810,159.833
C08092=1017.937,298.086,-139.481,169.941,50.815,159.833
C08093=1017.930,297.839,-139.450,169.936,50.819,159.833
C08094=1017.924,297.590,-139.418,169.930,50.823,159.833
C08095=1017.918,297.344,-139.386,169.924,50.828,159.833
C08096=1017.912,297.096,-139.354,169.919,50.833,159.834
C08097=1017.905,296.848,-139.322,169.913,50.837,159.834
C08098=1017.899,296.599,-139.290,169.908,50.841,159.834
C08099=1017.893,296.352,-139.259,169.902,50.846,159.834
C08100=1017.887,296.104,-139.227,169.896,50.850,159.834
C08101=1017.881,295.856,-139.195,169.891,50.855,159.834
C08102=1017.875,295.608,-139.165,169.886,50.859,159.834
C08103=1017.869,295.360,-139.133,169.880,50.864,159.834
C08104=1017.862,295.112,-139.101,169.875,50.869,159.834
C08105=1017.857,294.864,-139.070,169.869,50.873,159.834
C08106=1017.850,294.616,-139.038,169.863,50.878,159.834
C08107=1017.844,294.368,-139.006,169.859,50.882,159.834
C08108=1017.838,294.121,-138.975,169.853,50.887,159.834
C08109=1017.832,293.881,-138.944,169.847,50.891,159.834
C08110=1017.827,293.640,-138.913,169.842,50.895,159.834
C08111=1017.821,293.400,-138.884,169.837,50.900,159.835
C08112=1017.815,293.160,-138.853,169.832,50.904,159.835
C08113=1017.809,292.919,-138.822,169.826,50.909,159.835
C08114=1017.803,292.680,-138.792,169.822,50.913,159.835
C08115=1017.797,292.439,-138.762,169.816,50.918,159.835
C08116=1017.791,292.199,-138.733,169.810,50.923,159.835
C08117=1017.785,291.951,-138.701,169.806,50.927,159.835
C08118=1017.778,291.703,-138.669,169.800,50.932,159.835
C08119=1017.772,291.455,-138.639,169.795,50.937,159.836
C08120=1017.766,291.207,-138.608,169.789,50.942,159.836
C08121=1017.760,290.960,-138.577,169.783,50.947,159.836
C08122=1017.753,290.712,-138.546,169.778,50.952,159.836
C08123=1017.748,290.464,-138.515,169.773,50.956,159.836
C08124=1017.742,290.215,-138.484,169.768,50.961,159.836
C08125=1017.736,289.968,-138.453,169.762,50.966,159.836
C08126=1017.729,289.719,-138.422,169.757,50.971,159.837
C08127=1017.723,289.472,-138.391,169.751,50.976,159.837
C08128=1017.717,289.224,-138.361,169.745,50.981,159.837
C08129=1017.710,288.975,-138.330,169.740,50.986,159.837
C08130=1017.704,288.728,-138.299,169.736,50.991,159.837
C08131=1017.698,288.479,-138.268,169.730,50.995,159.837
C08132=1017.692,288.232,-138.238,169.724,51.000,159.838
C08133=1017.686,287.984,-138.207,169.719,51.005,159.838
C08134=1017.679,287.736,-138.176,169.713,51.010,159.838
C08135=1017.673,287.488,-138.146,169.708,51.015,159.838
C08136=1017.667,287.239,-138.115,169.704,51.020,159.838
C08137=1017.661,286.992,-138.085,169.698,51.025,159.839
C08138=1017.655,286.743,-138.054,169.693,51.030,159.839
C08139=1017.649,286.496,-138.023,169.687,51.035,159.839
C08140=1017.642,286.247,-137.992,169.682,51.040,159.839
C08141=1017.636,286.000,-137.962,169.676,51.046,159.839
C08142=1017.631,285.752,-137.931,169.671,51.051,159.840
C08143=1017.624,285.503,-137.901,169.666,51.055,159.840
C08144=1017.618,285.255,-137.870,169.661,51.061,159.840
C08145=1017.612,285.007,-137.840,169.656,51.066,159.840
C08146=1017.606,284.759,-137.809,169.650,51.071,159.840
C08147=1017.600,284.511,-137.779,169.645,51.076,159.841
C08148=1017.594,284.263,-137.748,169.639,51.081,159.841
C08149=1017.587,284.015,-137.718,169.634,51.086,159.841
C08150=1017.582,283.767,-137.688,169.629,51.091,159.841
C08151=1017.575,283.519,-137.657,169.624,51.096,159.841
C08152=1017.569,283.271,-137.627,169.619,51.102,159.842
C08153=1017.563,283.024,-137.597,169.614,51.107,159.842
C08154=1017.557,282.774,-137.567,169.608,51.112,159.842
C08155=1017.551,282.527,-137.537,169.603,51.117,159.842
C08156=1017.545,282.279,-137.507,169.597,51.122,159.843
C08157=1017.538,282.031,-137.476,169.592,51.128,159.843
C08158=1017.532,281.783,-137.446,169.587,51.133,159.843
C08159=1017.527,281.534,-137.416,169.582,51.138,159.843
C08160=1017.521,281.286,-137.386,169.577,51.144,159.844
C08161=1017.514,281.038,-137.356,169.572,51.149,159.844
C08162=1017.508,280.790,-137.326,169.566,51.154,159.844
C08163=1017.502,280.542,-137.296,169.561,51.160,159.845
C08164=1017.496,280.294,-137.266,169.556,51.165,159.845
C08165=1017.489,280.046,-137.236,169.551,51.170,159.845
C08166=1017.484,279.798,-137.206,169.546,51.176,159.845
C08167=1017.478,279.550,-137.176,169.540,51.181,159.846
C08168=1017.472,279.302,-137.145,169.536,51.186,159.846
C08169=1017.466,279.067,-137.117,169.531,51.191,159.846
C08170=1017.461,278.833,-137.089,169.526,51.196,159.846
C08171=1017.455,278.600,-137.061,169.521,51.201,159.847
C08172=1017.449,278.365,-137.032,169.516,51.206,159.847
C08173=1017.443,278.131,-137.005,169.511,51.211,159.847
C08174=1017.438,277.897,-136.976,169.507,51.217,159.848
C08175=1017.433,277.663,-136.947,169.501,51.222,159.848
C08176=1017.427,277.429,-136.920,169.497,51.226,159.848
C08177=1017.421,277.181,-136.889,169.492,51.232,159.848
C08178=1017.415,276.933,-136.860,169.487,51.237,159.849
C08179=1017.409,276.685,-136.830,169.482,51.243,159.849
C08180=1017.403,276.437,-136.800,169.476,51.248,159.849
C08181=1017.397,276.188,-136.770,169.471,51.254,159.850
C08182=1017.391,275.940,-136.741,169.466,51.259,159.850
C08183=1017.385,275.692,-136.711,169.461,51.265,159.850
C08184=1017.379,275.444,-136.681,169.456,51.271,159.851
C08185=1017.372,275.196,-136.652,169.451,51.277,159.851
C08186=1017.367,274.947,-136.622,169.445,51.282,159.851
C08187=1017.360,274.700,-136.593,169.440,51.288,159.852
C08188=1017.355,274.452,-136.563,169.436,51.293,159.852
C08189=1017.349,274.203,-136.534,169.431,51.298,159.852
C08190=1017.343,273.955,-136.504,169.426,51.304,159.853
C08191=1017.336,273.707,-136.475,169.421,51.310,159.853
C08192=1017.331,273.459,-136.445,169.416,51.316,159.853
C08193=1017.325,273.211,-136.416,169.411,51.321,159.854
C08194=1017.319,272.962,-136.386,169.405,51.327,159.854
C08195=1017.313,272.714,-136.357,169.400,51.332,159.854
C08196=1017.307,272.466,-136.327,169.395,51.338,159.855
C08197=1017.301,272.218,-136.298,169.390,51.344,159.855
C08198=1017.295,271.970,-136.268,169.385,51.350,159.856
C08199=1017.289,271.722,-136.239,169.380,51.356,159.856
C08200=1017.283,271.474,-136.210,169.375,51.361,159.856
C08201=1017.277,271.225,-136.181,169.370,51.367,159.856
C08202=1017.271,270.977,-136.152,169.365,51.372,159.857
C08203=1017.266,270.729,-136.122,169.360,51.378,159.857
C08204=1017.259,270.480,-136.093,169.355,51.384,159.858
C08205=1017.253,270.232,-136.064,169.350,51.390,159.858
C08206=1017.248,269.984,-136.034,169.345,51.396,159.858
C08207=1017.241,269.736,-136.005,169.340,51.402,159.859
C08208=1017.236,269.487,-135.975,169.335,51.407,159.859
C08209=1017.230,269.239,-135.946,169.330,51.413,159.860
C08210=1017.224,268.992,-135.918,169.325,51.419,159.860
C08211=1017.218,268.743,-135.888,169.320,51.426,159.861
C08212=1017.212,268.495,-135.859,169.315,51.431,159.861
C08213=1017.206,268.246,-135.831,169.310,51.437,159.861
C08214=1017.200,267.998,-135.802,169.305,51.443,159.862
C08215=1017.194,267.750,-135.773,169.300,51.449,159.862
C08216=1017.188,267.502,-135.743,169.295,51.455,159.863
C08217=1017.183,267.254,-135.714,169.290,51.461,159.863
C08218=1017.177,267.006,-135.686,169.286,51.467,159.863
C08219=1017.170,266.757,-135.657,169.281,51.473,159.864
C08220=1017.165,266.509,-135.627,169.276,51.479,159.864
C08221=1017.159,266.260,-135.599,169.271,51.485,159.865
C08222=1017.153,266.012,-135.570,169.266,51.491,159.865
C08223=1017.147,265.765,-135.541,169.261,51.497,159.866
C08224=1017.141,265.517,-135.512,169.256,51.503,159.866
C08225=1017.136,265.267,-135.483,169.251,51.509,159.866
C08226=1017.129,265.019,-135.454,169.247,51.515,159.867
C08227=1017.123,264.771,-135.426,169.242,51.521,159.867
C08228=1017.118,264.523,-135.397,169.237,51.527,159.868
C08229=1017.112,264.291,-135.371,169.233,51.532,159.868
C08230=1017.106,264.059,-135.343,169.228,51.539,159.869
C08231=1017.101,263.827,-135.317,169.223,51.545,159.869
C08232=1017.095,263.595,-135.291,169.219,51.550,159.870
C08233=1017.090,263.364,-135.263,169.214,51.556,159.870
C08234=1017.084,263.132,-135.237,169.210,51.561,159.871
C08235=1017.079,262.900,-135.211,169.205,51.567,159.871
C08236=1017.073,262.669,-135.183,169.200,51.573,159.871
C08237=1017.067,262.420,-135.155,169.195,51.579,159.872
C08238=1017.061,262.172,-135.126,169.191,51.586,159.872
C08239=1017.056,261.924,-135.098,169.186,51.591,159.873
C08240=1017.050,261.675,-135.070,169.181,51.598,159.873
C08241=1017.044,261.427,-135.041,169.176,51.604,159.874
C08242=1017.038,261.179,-135.013,169.171,51.610,159.874
C08243=1017.032,260.931,-134.984,169.167,51.617,159.875
C08244=1017.027,260.682,-134.955,169.162,51.623,159.875
C08245=1017.021,260.434,-134.927,169.157,51.629,159.876
C08246=1017.015,260.185,-134.898,169.152,51.635,159.876
C08247=1017.009,259.937,-134.870,169.148,51.642,159.877
C08248=1017.004,259.689,-134.842,169.143,51.648,159.877
C08249=1016.997,259.440,-134.814,169.137,51.654,159.878
C08250=1016.991,259.191,-134.785,169.133,51.661,159.878
C08251=1016.986,258.943,-134.758,169.128,51.667,159.879
C08252=1016.979,258.696,-134.729,169.124,51.674,159.880
C08253=1016.973,258.447,-134.701,169.119,51.681,159.880
C08254=1016.967,258.199,-134.673,169.114,51.687,159.881
C08255=1016.961,257.950,-134.645,169.108,51.693,159.881
C08256=1016.955,257.702,-134.617,169.104,51.700,159.882
C08257=1016.949,257.454,-134.589,169.099,51.706,159.882
C08258=1016.943,257.205,-134.561,169.095,51.713,159.883
C08259=1016.938,256.957,-134.533,169.090,51.720,159.883
C08260=1016.931,256.709,-134.505,169.085,51.726,159.884
C08261=1016.925,256.460,-134.477,169.080,51.733,159.884
C08262=1016.919,256.212,-134.450,169.076,51.740,159.885
C08263=1016.913,255.963,-134.422,169.071,51.746,159.886
C08264=1016.908,255.715,-134.394,169.066,51.753,159.886
C08265=1016.901,255.466,-134.366,169.061,51.760,159.887
C08266=1016.896,255.218,-134.338,169.056,51.766,159.887
C08267=1016.890,254.969,-134.310,169.052,51.773,159.888
C08268=1016.884,254.722,-134.283,169.047,51.779,159.889
C08269=1016.878,254.473,-134.254,169.043,51.786,159.889
C08270=1016.872,254.224,-134.226,169.037,51.793,159.890
C08271=1016.866,253.976,-134.199,169.033,51.799,159.890
C08272=1016.860,253.727,-134.171,169.028,51.806,159.891
C08273=1016.854,253.479,-134.144,169.023,51.812,159.891
C08274=1016.849,253.231,-134.116,169.019,51.819,159.892
C08275=1016.843,252.982,-134.087,169.013,51.826,159.893
C08276=1016.837,252.735,-134.060,169.009,51.832,159.893
C08277=1016.831,252.485,-134.032,169.004,51.839,159.894
C08278=1016.826,252.237,-134.005,169.000,51.846,159.894
C08279=1016.819,251.989,-133.977,168.996,51.853,159.895
C08280=1016.814,251.741,-133.949,168.990,51.860,159.896
C08281=1016.808,251.492,-133.922,168.986,51.866,159.896
C08282=1016.802,251.244,-133.894,168.981,51.873,159.897
C08283=1016.797,250.996,-133.866,168.976,51.879,159.897
C08284=1016.790,250.747,-133.839,168.971,51.887,159.898
C08285=1016.785,250.499,-133.811,168.967,51.894,159.899
C08286=1016.778,250.250,-133.783,168.962,51.900,159.899
C08287=1016.773,250.001,-133.756,168.958,51.907,159.900
C08288=1016.768,249.753,-133.728,168.952,51.914,159.900
C08289=1016.762,249.520,-133.702,168.949,51.920,159.901
C08290=1016.757,249.288,-133.677,168.944,51.927,159.902
C08291=1016.752,249.055,-133.651,168.940,51.933,159.902
C08292=1016.747,248.823,-133.625,168.935,51.940,159.903
C08293=1016.741,248.590,-133.599,168.932,51.946,159.904
C08294=1016.736,248.357,-133.573,168.927,51.953,159.904
C08295=1016.730,248.125,-133.547,168.923,51.959,159.905
C08296=1016.725,247.891,-133.521,168.918,51.966,159.905
C08297=1016.719,247.643,-133.494,168.913,51.972,159.906
C08298=1016.714,247.395,-133.466,168.909,51.979,159.906
C08299=1016.708,247.147,-133.440,168.905,51.986,159.907
C08300=1016.702,246.898,-133.412,168.899,51.993,159.908
C08301=1016.697,246.649,-133.384,168.895,52.000,159.909
C08302=1016.691,246.402,-133.357,168.891,52.007,159.909
C08303=1016.686,246.153,-133.330,168.886,52.014,159.910
C08304=1016.680,245.904,-133.301,168.881,52.021,159.910
C08305=1016.674,245.656,-133.275,168.877,52.028,159.911
C08306=1016.669,245.408,-133.247,168.872,52.035,159.912
C08307=1016.663,245.159,-133.220,168.867,52.042,159.912
C08308=1016.657,244.910,-133.192,168.863,52.049,159.913
C08309=1016.652,244.662,-133.165,168.858,52.056,159.914
C08310=1016.646,244.414,-133.138,168.854,52.063,159.915
C08311=1016.641,244.166,-133.110,168.849,52.070,159.915
C08312=1016.635,243.917,-133.083,168.845,52.078,159.916
C08313=1016.630,243.668,-133.056,168.840,52.084,159.916
C08314=1016.624,243.420,-133.028,168.836,52.091,159.917
C08315=1016.618,243.171,-133.001,168.831,52.098,159.918
C08316=1016.613,242.923,-132.974,168.826,52.106,159.919
C08317=1016.607,242.675,-132.946,168.822,52.113,159.919
C08318=1016.601,242.426,-132.919,168.817,52.120,159.920
C08319=1016.596,242.177,-132.892,168.813,52.127,159.921
C08320=1016.590,241.929,-132.866,168.809,52.135,159.921
C08321=1016.584,241.681,-132.839,168.803,52.142,159.922
C08322=1016.579,241.432,-132.812,168.799,52.149,159.923
C08323=1016.574,241.183,-132.785,168.794,52.157,159.923
C08324=1016.567,240.934,-132.758,168.790,52.164,159.924
C08325=1016.562,240.686,-132.730,168.786,52.171,159.925
C08326=1016.556,240.438,-132.703,168.780,52.178,159.926
C08327=1016.550,240.190,-132.677,168.776,52.185,159.926
C08328=1016.545,239.941,-132.649,168.772,52.193,159.927
C08329=1016.539,239.693,-132.623,168.767,52.200,159.928
C08330=1016.534,239.444,-132.596,168.763,52.208,159.929
C08331=1016.528,239.196,-132.570,168.758,52.215,159.929
C08332=1016.523,238.947,-132.542,168.754,52.222,159.930
C08333=1016.517,238.699,-132.516,168.750,52.229,159.931
C08334=1016.511,238.451,-132.489,168.744,52.237,159.931
C08335=1016.506,238.202,-132.462,168.740,52.244,159.932
C08336=1016.500,237.954,-132.436,168.735,52.252,159.933
C08337=1016.494,237.704,-132.409,168.731,52.259,159.934
C08338=1016.488,237.456,-132.383,168.726,52.267,159.934
C08339=1016.482,237.207,-132.356,168.723,52.275,159.936
C08340=1016.476,236.959,-132.329,168.718,52.283,159.936
C08341=1016.471,236.711,-132.303,168.713,52.290,159.937
C08342=1016.465,236.462,-132.277,168.708,52.298,159.938
C08343=1016.459,236.213,-132.250,168.704,52.305,159.939
C08344=1016.454,235.965,-132.224,168.699,52.313,159.939
C08345=1016.448,235.717,-132.197,168.695,52.320,159.940
C08346=1016.442,235.468,-132.171,168.690,52.328,159.941
C08347=1016.437,235.219,-132.144,168.687,52.336,159.942
C08348=1016.431,234.971,-132.118,168.682,52.344,159.942
C08349=1016.426,234.735,-132.093,168.677,52.351,159.943
C08350=1016.420,234.499,-132.067,168.673,52.358,159.944
C08351=1016.415,234.263,-132.043,168.669,52.365,159.945
C08352=1016.410,234.027,-132.018,168.665,52.372,159.945
C08353=1016.404,233.791,-131.993,168.661,52.380,159.946
C08354=1016.399,233.555,-131.967,168.656,52.387,159.947
C08355=1016.393,233.318,-131.943,168.652,52.395,159.948
C08356=1016.388,233.082,-131.918,168.648,52.402,159.949
C08357=1016.383,232.834,-131.891,168.643,52.410,159.949
C08358=1016.377,232.586,-131.864,168.639,52.417,159.950
C08359=1016.371,232.337,-131.838,168.634,52.425,159.951
C08360=1016.366,232.088,-131.812,168.630,52.433,159.952
C08361=1016.360,231.839,-131.786,168.625,52.440,159.953
C08362=1016.354,231.591,-131.759,168.621,52.448,159.954
C08363=1016.349,231.342,-131.733,168.616,52.456,159.954
C08364=1016.344,231.094,-131.707,168.613,52.464,159.955
C08365=1016.338,230.845,-131.681,168.608,52.472,159.956
C08366=1016.332,230.597,-131.655,168.603,52.480,159.957
C08367=1016.326,230.348,-131.629,168.599,52.488,159.958
C08368=1016.321,230.100,-131.602,168.594,52.495,159.958
C08369=1016.315,229.851,-131.577,168.591,52.504,159.959
C08370=1016.309,229.602,-131.550,168.585,52.511,159.960
C08371=1016.304,229.354,-131.524,168.581,52.520,159.961
C08372=1016.299,229.106,-131.498,168.577,52.527,159.962
C08373=1016.293,228.857,-131.472,168.572,52.535,159.963
C08374=1016.287,228.608,-131.446,168.568,52.543,159.964
C08375=1016.281,228.360,-131.420,168.564,52.551,159.965
C08376=1016.276,228.111,-131.394,168.559,52.559,159.965
C08377=1016.271,227.863,-131.368,168.555,52.567,159.966
C08378=1016.265,227.614,-131.342,168.551,52.575,159.967
C08379=1016.259,227.366,-131.316,168.546,52.583,159.968
C08380=1016.253,227.117,-131.290,168.542,52.591,159.969
C08381=1016.248,226.868,-131.264,168.537,52.600,159.970
C08382=1016.243,226.620,-131.238,168.532,52.607,159.970
C08383=1016.237,226.371,-131.212,168.529,52.616,159.972
C08384=1016.231,226.122,-131.187,168.524,52.624,159.972
C08385=1016.226,225.873,-131.161,168.519,52.632,159.973
C08386=1016.220,225.625,-131.136,168.516,52.640,159.974
C08387=1016.215,225.376,-131.110,168.511,52.648,159.975
C08388=1016.209,225.127,-131.084,168.507,52.657,159.976
C08389=1016.203,224.879,-131.059,168.502,52.665,159.977
C08390=1016.198,224.630,-131.033,168.497,52.674,159.978
C08391=1016.192,224.382,-131.007,168.493,52.681,159.979
C08392=1016.186,224.133,-130.981,168.489,52.689,159.980
C08393=1016.180,223.885,-130.956,168.484,52.698,159.981
C08394=1016.175,223.636,-130.930,168.480,52.706,159.981
C08395=1016.169,223.388,-130.905,168.476,52.714,159.982
C08396=1016.163,223.139,-130.879,168.472,52.723,159.983
C08397=1016.158,222.890,-130.853,168.467,52.731,159.984
C08398=1016.152,222.642,-130.828,168.463,52.740,159.985
C08399=1016.147,222.393,-130.802,168.458,52.748,159.986
C08400=1016.141,222.144,-130.778,168.454,52.756,159.987
C08401=1016.136,221.895,-130.752,168.450,52.765,159.988
C08402=1016.130,221.647,-130.727,168.445,52.773,159.989
C08403=1016.124,221.398,-130.701,168.441,52.782,159.990
C08404=1016.119,221.150,-130.676,168.436,52.790,159.991
C08405=1016.113,220.901,-130.650,168.433,52.798,159.992
C08406=1016.108,220.652,-130.624,168.428,52.807,159.993
C08407=1016.102,220.404,-130.599,168.424,52.815,159.994
C08408=1016.097,220.155,-130.573,168.419,52.824,159.995
C08409=1016.091,219.915,-130.549,168.416,52.832,159.996
C08410=1016.086,219.675,-130.524,168.411,52.840,159.997
C08411=1016.081,219.434,-130.500,168.406,52.848,159.997
C08412=1016.075,219.194,-130.475,168.403,52.856,159.998
C08413=1016.070,218.954,-130.451,168.398,52.865,159.999
C08414=1016.065,218.714,-130.426,168.395,52.873,160.000
C08415=1016.059,218.473,-130.402,168.390,52.881,160.001
C08416=1016.054,218.233,-130.377,168.387,52.889,160.002
C08417=1016.048,217.984,-130.352,168.382,52.898,160.003
C08418=1016.043,217.736,-130.327,168.378,52.906,160.004
C08419=1016.037,217.487,-130.301,168.373,52.916,160.005
C08420=1016.032,217.239,-130.277,168.369,52.924,160.006
C08421=1016.026,216.990,-130.251,168.364,52.933,160.007
C08422=1016.020,216.741,-130.227,168.360,52.942,160.008
C08423=1016.015,216.492,-130.201,168.356,52.950,160.009
C08424=1016.009,216.244,-130.176,168.351,52.959,160.010
C08425=1016.003,215.995,-130.152,168.347,52.968,160.011
C08426=1015.997,215.746,-130.126,168.343,52.976,160.012
C08427=1015.993,215.498,-130.101,168.339,52.986,160.013
C08428=1015.986,215.249,-130.076,168.334,52.994,160.014
C08429=1015.981,215.000,-130.052,168.330,53.003,160.015
C08430=1015.975,214.752,-130.027,168.326,53.012,160.016
C08431=1015.970,214.503,-130.002,168.321,53.020,160.017
C08432=1015.964,214.254,-129.976,168.317,53.030,160.018
C08433=1015.959,214.006,-129.952,168.313,53.038,160.019
C08434=1015.953,213.757,-129.927,168.309,53.047,160.020
C08435=1015.948,213.508,-129.902,168.304,53.056,160.021
C08436=1015.942,213.259,-129.877,168.300,53.065,160.023
C08437=1015.937,213.011,-129.852,168.296,53.074,160.023
C08438=1015.931,212.763,-129.827,168.292,53.083,160.025
C08439=1015.926,212.513,-129.802,168.287,53.092,160.026
C08440=1015.920,212.265,-129.777,168.283,53.100,160.027
C08441=1015.914,212.016,-129.753,168.279,53.110,160.028
C08442=1015.909,211.767,-129.728,168.274,53.118,160.029
C08443=1015.904,211.518,-129.702,168.270,53.127,160.030
C08444=1015.898,211.270,-129.678,168.266,53.137,160.031
C08445=1015.893,211.022,-129.653,168.262,53.145,160.032
C08446=1015.887,210.772,-129.629,168.258,53.154,160.033
C08447=1015.881,210.524,-129.604,168.254,53.164,160.034
C08448=1015.876,210.275,-129.578,168.249,53.172,160.035
C08449=1015.871,210.026,-129.554,168.244,53.182,160.036
C08450=1015.865,209.778,-129.530,168.240,53.191,160.037
C08451=1015.859,209.529,-129.504,168.236,53.200,160.038
C08452=1015.854,209.280,-129.480,168.232,53.209,160.039
C08453=1015.849,209.032,-129.456,168.228,53.218,160.041
C08454=1015.843,208.782,-129.431,168.224,53.227,160.042
C08455=1015.838,208.534,-129.406,168.220,53.237,160.043
C08456=1015.832,208.285,-129.381,168.215,53.245,160.044
C08457=1015.827,208.036,-129.357,168.210,53.255,160.045
C08458=1015.821,207.788,-129.333,168.206,53.264,160.046
C08459=1015.815,207.539,-129.308,168.202,53.273,160.047
C08460=1015.810,207.290,-129.284,168.198,53.283,160.048
C08461=1015.805,207.041,-129.259,168.195,53.292,160.050
C08462=1015.800,206.793,-129.235,168.189,53.301,160.051
C08463=1015.793,206.544,-129.210,168.186,53.311,160.052
C08464=1015.788,206.296,-129.186,168.182,53.320,160.053
C08465=1015.783,206.047,-129.161,168.178,53.329,160.054
C08466=1015.777,205.798,-129.137,168.173,53.339,160.055
C08467=1015.772,205.549,-129.113,168.169,53.348,160.056
C08468=1015.765,205.301,-129.089,168.165,53.357,160.057
C08469=1015.760,205.064,-129.065,168.160,53.366,160.058
C08470=1015.755,204.829,-129.043,168.156,53.375,160.059
C08471=1015.750,204.593,-129.020,168.152,53.384,160.061
C08472=1015.745,204.357,-128.996,168.149,53.393,160.062
C08473=1015.739,204.121,-128.973,168.145,53.402,160.063
C08474=1015.734,203.885,-128.951,168.141,53.411,160.064
C08475=1015.729,203.650,-128.928,168.137,53.421,160.065
C08476=1015.723,203.413,-128.905,168.132,53.429,160.066
C08477=1015.701,202.198,-128.795,167.622,53.370,159.946
C08478=1015.697,201.954,-128.773,167.617,53.381,159.947
C08479=1015.693,201.711,-128.750,167.611,53.391,159.948
C08480=1015.688,201.468,-128.729,167.607,53.402,159.949
C08481=1015.684,201.218,-128.706,167.602,53.412,159.950
C08482=1015.679,200.970,-128.683,167.598,53.423,159.952
C08483=1015.674,200.721,-128.661,167.593,53.434,159.953
C08484=1015.670,200.472,-128.639,167.589,53.444,159.954
C08485=1015.666,200.223,-128.617,167.584,53.455,159.955
C08486=1015.661,199.974,-128.595,167.579,53.466,159.957
C08487=1015.657,199.725,-128.571,167.574,53.476,159.958
C08488=1015.653,199.476,-128.549,167.570,53.487,159.959
C08489=1015.648,199.227,-128.527,167.566,53.498,159.960
C08490=1015.644,198.978,-128.505,167.560,53.509,159.961
C08491=1015.639,198.729,-128.482,167.556,53.520,159.963
C08492=1015.635,198.480,-128.460,167.551,53.530,159.964
C08493=1015.630,198.231,-128.438,167.546,53.541,159.965
C08494=1015.625,197.982,-128.416,167.542,53.552,159.967
C08495=1015.620,197.733,-128.394,167.537,53.562,159.968
C08496=1015.616,197.484,-128.372,167.533,53.574,159.969
C08497=1015.611,197.235,-128.350,167.527,53.584,159.970
C08498=1015.606,196.986,-128.328,167.523,53.596,159.972
C08499=1015.602,196.737,-128.306,167.519,53.606,159.973
C08500=1015.598,196.488,-128.285,167.514,53.617,159.974
C08501=1015.593,196.239,-128.263,167.509,53.628,159.975
C08502=1015.588,195.990,-128.241,167.505,53.639,159.977
C08503=1015.584,195.741,-128.218,167.501,53.650,159.978
C08504=1015.579,195.492,-128.197,167.495,53.661,159.979
C08505=1015.574,195.243,-128.175,167.491,53.671,159.980
C08506=1015.570,194.994,-128.152,167.487,53.683,159.982
C08507=1015.566,194.745,-128.131,167.482,53.693,159.983
C08508=1015.561,194.496,-128.109,167.478,53.704,159.984
C08509=1015.556,194.247,-128.087,167.473,53.715,159.986
C08510=1015.552,193.998,-128.065,167.469,53.726,159.987
C08511=1015.547,193.749,-128.043,167.464,53.737,159.988
C08512=1015.543,193.500,-128.022,167.460,53.748,159.990
C08513=1015.539,193.251,-127.999,167.455,53.758,159.991
C08514=1015.534,193.002,-127.978,167.450,53.769,159.992
C08515=1015.529,192.753,-127.956,167.446,53.780,159.993
C08516=1015.525,192.504,-127.935,167.441,53.791,159.994
C08517=1015.520,192.230,-127.911,167.437,53.803,159.996
C08518=1015.515,191.956,-127.886,167.432,53.815,159.997
C08519=1015.511,191.683,-127.862,167.427,53.827,159.999
C08520=1015.505,191.409,-127.838,167.422,53.839,160.000
C08521=1015.501,191.160,-127.817,167.418,53.850,160.002
C08522=1015.496,190.911,-127.795,167.413,53.860,160.003
C08523=1015.493,190.662,-127.773,167.408,53.872,160.004
C08524=1015.488,190.413,-127.752,167.404,53.882,160.005
C08525=1015.483,190.164,-127.730,167.400,53.893,160.007
C08526=1015.478,189.915,-127.708,167.395,53.904,160.008
C08527=1015.475,189.665,-127.686,167.391,53.915,160.009
C08528=1015.470,189.417,-127.664,167.387,53.926,160.010
C08529=1015.466,189.168,-127.644,167.383,53.937,160.012
C08530=1015.461,188.919,-127.622,167.378,53.947,160.013
C08531=1015.457,188.670,-127.599,167.374,53.959,160.014
C08532=1015.452,188.421,-127.578,167.370,53.969,160.016
C08533=1015.448,188.172,-127.556,167.365,53.980,160.017
C08534=1015.444,187.923,-127.535,167.360,53.991,160.018
C08535=1015.440,187.674,-127.513,167.356,54.002,160.019
C08536=1015.435,187.424,-127.492,167.352,54.013,160.021
C08537=1015.430,187.145,-127.467,167.347,54.025,160.022
C08538=1015.425,186.865,-127.443,167.342,54.037,160.024
C08539=1015.421,186.585,-127.419,167.338,54.049,160.025
C08540=1015.416,186.305,-127.395,167.333,54.062,160.027
C08541=1015.412,186.057,-127.373,167.329,54.072,160.028
C08542=1015.407,185.807,-127.352,167.325,54.083,160.029
C08543=1015.402,185.559,-127.330,167.320,54.094,160.031
C08544=1015.398,185.309,-127.308,167.316,54.104,160.032
C08545=1015.394,185.061,-127.287,167.312,54.116,160.033
C08546=1015.390,184.811,-127.266,167.308,54.126,160.034
C08547=1015.386,184.562,-127.243,167.304,54.137,160.036
C08548=1015.382,184.313,-127.223,167.299,54.148,160.037
C08549=1015.377,184.065,-127.201,167.295,54.159,160.038
C08550=1015.372,183.815,-127.180,167.291,54.170,160.040
C08551=1015.369,183.566,-127.158,167.286,54.180,160.041
C08552=1015.364,183.317,-127.136,167.282,54.192,160.042
C08553=1015.360,183.068,-127.115,167.278,54.202,160.043
C08554=1015.356,182.819,-127.094,167.274,54.213,160.045
C08555=1015.352,182.570,-127.072,167.270,54.224,160.046
C08556=1015.347,182.321,-127.051,167.265,54.235,160.047
C08557=1015.343,182.072,-127.030,167.261,54.246,160.049
C08558=1015.339,181.823,-127.008,167.257,54.256,160.050
C08559=1015.335,181.573,-126.986,167.253,54.268,160.051
C08560=1015.330,181.324,-126.966,167.249,54.278,160.053
C08561=1015.326,181.075,-126.945,167.245,54.290,160.054
C08562=1015.321,180.826,-126.924,167.241,54.301,160.055
C08563=1015.316,180.577,-126.903,167.237,54.312,160.057
C08564=1015.312,180.328,-126.883,167.232,54.323,160.058
C08565=1015.307,180.079,-126.862,167.229,54.334,160.059
C08566=1015.303,179.830,-126.841,167.224,54.346,160.061
C08567=1015.298,179.581,-126.820,167.220,54.357,160.062
C08568=1015.293,179.331,-126.800,167.215,54.368,160.063
C08569=1015.289,179.082,-126.780,167.211,54.379,160.065
C08570=1015.284,178.833,-126.759,167.208,54.390,160.066
C08571=1015.280,178.584,-126.738,167.204,54.402,160.068
C08572=1015.276,178.335,-126.717,167.199,54.412,160.069
C08573=1015.270,178.086,-126.696,167.195,54.423,160.070
C08574=1015.267,177.837,-126.676,167.192,54.435,160.072
C08575=1015.261,177.588,-126.655,167.187,54.445,160.073
C08576=1015.258,177.339,-126.635,167.183,54.457,160.075
C08577=1015.253,177.089,-126.614,167.179,54.468,160.076
C08578=1015.248,176.840,-126.593,167.175,54.479,160.077
C08579=1015.244,176.591,-126.573,167.170,54.490,160.078
C08580=1015.239,176.342,-126.552,167.166,54.502,160.080
C08581=1015.235,176.094,-126.531,167.162,54.513,160.081
C08582=1015.231,175.844,-126.511,167.158,54.524,160.083
C08583=1015.226,175.595,-126.491,167.154,54.535,160.084
C08584=1015.221,175.346,-126.469,167.150,54.546,160.085
C08585=1015.217,175.097,-126.449,167.146,54.557,160.087
C08586=1015.212,174.848,-126.428,167.142,54.568,160.088
C08587=1015.209,174.599,-126.408,167.138,54.580,160.090
C08588=1015.203,174.349,-126.388,167.134,54.590,160.091
C08589=1015.199,174.101,-126.367,167.130,54.602,160.092
C08590=1015.195,173.851,-126.347,167.126,54.613,160.094
C08591=1015.191,173.602,-126.326,167.122,54.624,160.095
C08592=1015.186,173.353,-126.305,167.118,54.635,160.096
C08593=1015.181,173.104,-126.285,167.114,54.646,160.098
C08594=1015.177,172.854,-126.264,167.111,54.657,160.099
C08595=1015.173,172.606,-126.244,167.107,54.668,160.101
C08596=1015.168,172.356,-126.223,167.103,54.679,160.102
C08597=1015.164,172.107,-126.203,167.099,54.690,160.103
C08598=1015.159,171.858,-126.182,167.095,54.701,160.105
C08599=1015.155,171.609,-126.162,167.092,54.713,160.106
C08600=1015.151,171.360,-126.142,167.087,54.723,160.107
C08601=1015.146,171.080,-126.118,167.083,54.736,160.109
C08602=1015.141,170.800,-126.096,167.079,54.748,160.110
C08603=1015.137,170.520,-126.073,167.074,54.761,160.112
C08604=1015.131,170.240,-126.050,167.070,54.773,160.114
C08605=1015.127,169.991,-126.029,167.066,54.785,160.115
C08606=1015.122,169.742,-126.009,167.062,54.795,160.116
C08607=1015.118,169.493,-125.989,167.058,54.807,160.118
C08608=1015.115,169.244,-125.968,167.054,54.818,160.119
C08609=1015.110,168.994,-125.948,167.050,54.829,160.120
C08610=1015.106,168.745,-125.927,167.047,54.840,160.122
C08611=1015.101,168.496,-125.908,167.044,54.851,160.123
C08612=1015.097,168.247,-125.887,167.039,54.862,160.125
C08613=1015.092,167.998,-125.866,167.036,54.873,160.126
C08614=1015.089,167.749,-125.846,167.031,54.884,160.127
C08615=1015.084,167.500,-125.825,167.028,54.895,160.129
C08616=1015.080,167.251,-125.806,167.025,54.906,160.130
C08617=1015.076,167.002,-125.785,167.021,54.917,160.132
C08618=1015.071,166.752,-125.765,167.017,54.929,160.133
C08619=1015.067,166.503,-125.744,167.013,54.939,160.134
C08620=1015.063,166.254,-125.724,167.009,54.951,160.136
C08621=1015.058,166.005,-125.704,167.005,54.961,160.137
C08622=1015.054,165.756,-125.684,167.002,54.972,160.139
C08623=1015.050,165.507,-125.664,166.998,54.984,160.140
C08624=1015.046,165.257,-125.643,166.994,54.995,160.141
C08625=1015.041,165.008,-125.623,166.990,55.006,160.143
C08626=1015.037,164.759,-125.603,166.987,55.016,160.144
C08627=1015.034,164.510,-125.583,166.983,55.028,160.146
C08628=1015.028,164.261,-125.562,166.979,55.038,160.147
C08629=1015.025,164.012,-125.542,166.975,55.050,160.148
C08630=1015.020,163.762,-125.523,166.971,55.061,160.149
C08631=1015.017,163.514,-125.502,166.968,55.072,160.151
C08632=1015.012,163.264,-125.482,166.964,55.082,160.152
C08633=1015.008,163.015,-125.461,166.961,55.094,160.154
C08634=1015.004,162.766,-125.441,166.958,55.105,160.155
C08635=1015.000,162.517,-125.422,166.954,55.116,160.157
C08636=1014.995,162.267,-125.400,166.950,55.127,160.158
C08637=1014.991,162.018,-125.381,166.946,55.138,160.159
C08638=1014.987,161.769,-125.361,166.943,55.149,160.161
C08639=1014.983,161.520,-125.340,166.939,55.160,160.162
C08640=1014.979,161.271,-125.321,166.935,55.171,160.164
C08641=1014.975,161.021,-125.300,166.932,55.182,160.165
C08642=1014.970,160.773,-125.280,166.928,55.193,160.166
C08643=1014.966,160.523,-125.260,166.924,55.204,160.168
C08644=1014.962,160.274,-125.241,166.922,55.215,160.169
C08645=1014.958,160.026,-125.220,166.917,55.226,160.170
C08646=1014.955,159.776,-125.200,166.913,55.236,160.172
C08647=1014.950,159.527,-125.180,166.911,55.247,160.173
C08648=1014.946,159.278,-125.159,166.906,55.258,160.175
C08649=1014.941,159.029,-125.140,166.903,55.270,160.176
C08650=1014.938,158.779,-125.120,166.900,55.280,160.177
C08651=1014.934,158.530,-125.099,166.896,55.292,160.179
C08652=1014.929,158.280,-125.080,166.892,55.302,160.180
C08653=1014.925,158.031,-125.060,166.889,55.313,160.182
C08654=1014.921,157.782,-125.041,166.886,55.325,160.183
C08655=1014.916,157.533,-125.021,166.882,55.336,160.184
C08656=1014.913,157.284,-125.001,166.878,55.347,160.186
C08657=1014.908,157.035,-124.982,166.874,55.359,160.187
C08658=1014.903,156.785,-124.962,166.871,55.369,160.189
C08659=1014.899,156.536,-124.942,166.868,55.381,160.190
C08660=1014.895,156.287,-124.923,166.864,55.392,160.192
C08661=1014.890,156.038,-124.903,166.860,55.403,160.193
C08662=1014.886,155.789,-124.884,166.857,55.414,160.195
C08663=1014.882,155.540,-124.864,166.854,55.426,160.196
C08664=1014.877,155.291,-124.845,166.849,55.436,160.197
C08665=1014.872,155.010,-124.823,166.845,55.449,160.199
C08666=1014.868,154.730,-124.801,166.841,55.462,160.200
C08667=1014.862,154.450,-124.779,166.838,55.474,160.202
C08668=1014.858,154.169,-124.757,166.834,55.487,160.204
C08669=1014.853,153.920,-124.738,166.830,55.498,160.205
C08670=1014.849,153.671,-124.718,166.826,55.509,160.207
C08671=1014.845,153.422,-124.700,166.824,55.520,160.208
C08672=1014.841,153.173,-124.680,166.820,55.532,160.210
C08673=1014.837,152.923,-124.660,166.816,55.542,160.211
C08674=1014.833,152.674,-124.641,166.814,55.553,160.213
C08675=1014.828,152.425,-124.621,166.810,55.565,160.214
C08676=1014.824,152.175,-124.602,166.806,55.576,160.215
C08677=1014.819,151.926,-124.582,166.803,55.587,160.217
C08678=1014.815,151.677,-124.563,166.800,55.599,160.218
C08679=1014.810,151.428,-124.544,166.796,55.609,160.220
C08680=1014.806,151.178,-124.525,166.792,55.621,160.221
C08681=1014.802,150.929,-124.506,166.790,55.632,160.223
C08682=1014.797,150.680,-124.486,166.786,55.643,160.224
C08683=1014.793,150.431,-124.467,166.782,55.654,160.225
C08684=1014.789,150.181,-124.448,166.779,55.665,160.227
C08685=1014.785,149.932,-124.429,166.776,55.677,160.228
C08686=1014.780,149.683,-124.409,166.772,55.688,160.230
C08687=1014.776,149.434,-124.390,166.769,55.699,160.231
C08688=1014.772,149.185,-124.371,166.765,55.710,160.233
C08689=1014.767,148.936,-124.352,166.762,55.722,160.234
C08690=1014.763,148.686,-124.333,166.759,55.732,160.236
C08691=1014.759,148.437,-124.313,166.755,55.744,160.237
C08692=1014.755,148.187,-124.295,166.751,55.755,160.238
C08693=1014.751,147.938,-124.275,166.749,55.766,160.240
C08694=1014.746,147.689,-124.256,166.745,55.777,160.242
C08695=1014.742,147.440,-124.237,166.741,55.788,160.243
C08696=1014.738,147.191,-124.218,166.739,55.799,160.244
C08697=1014.734,146.942,-124.200,166.735,55.810,160.246
C08698=1014.729,146.693,-124.180,166.732,55.821,160.247
C08699=1014.725,146.443,-124.161,166.729,55.833,160.249
C08700=1014.721,146.194,-124.142,166.725,55.844,160.250
C08701=1014.717,145.945,-124.122,166.722,55.855,160.252
C08702=1014.712,145.696,-124.104,166.718,55.866,160.253
C08703=1014.708,145.447,-124.085,166.715,55.878,160.254
C08704=1014.703,145.197,-124.066,166.712,55.889,160.256
C08705=1014.699,144.947,-124.047,166.708,55.900,160.257
C08706=1014.694,144.699,-124.028,166.705,55.911,160.259
C08707=1014.690,144.449,-124.010,166.703,55.922,160.261
C08708=1014.686,144.200,-123.990,166.699,55.933,160.262
C08709=1014.681,143.951,-123.972,166.696,55.945,160.263
C08710=1014.678,143.702,-123.954,166.693,55.956,160.265
C08711=1014.673,143.453,-123.934,166.689,55.967,160.266
C08712=1014.669,143.203,-123.916,166.686,55.978,160.268
C08713=1014.665,142.954,-123.897,166.682,55.989,160.269
C08714=1014.660,142.704,-123.878,166.679,56.001,160.271
C08715=1014.655,142.455,-123.860,166.676,56.012,160.272
C08716=1014.651,142.205,-123.841,166.672,56.023,160.274
C08717=1014.647,141.956,-123.821,166.670,56.034,160.275
C08718=1014.643,141.708,-123.804,166.666,56.045,160.277
C08719=1014.639,141.458,-123.785,166.663,56.057,160.278
C08720=1014.634,141.209,-123.765,166.660,56.068,160.280
C08721=1014.630,140.960,-123.747,166.656,56.079,160.281
C08722=1014.626,140.710,-123.728,166.654,56.090,160.283
C08723=1014.621,140.461,-123.710,166.650,56.101,160.284
C08724=1014.617,140.212,-123.691,166.647,56.113,160.285
C08725=1014.613,139.963,-123.672,166.644,56.123,160.287
C08726=1014.608,139.713,-123.654,166.640,56.135,160.288
C08727=1014.604,139.464,-123.635,166.638,56.146,160.290
C08728=1014.600,139.215,-123.616,166.634,56.157,160.291
C08729=1014.595,138.935,-123.595,166.631,56.169,160.293
C08730=1014.591,138.654,-123.574,166.627,56.182,160.295
C08731=1014.585,138.374,-123.553,166.624,56.195,160.297
C08732=1014.580,138.094,-123.533,166.620,56.207,160.298
C08733=1014.576,137.845,-123.513,166.617,56.218,160.299
C08734=1014.573,137.596,-123.495,166.614,56.229,160.301
C08735=1014.568,137.346,-123.477,166.610,56.241,160.302
C08736=1014.564,137.097,-123.458,166.608,56.252,160.304
C08737=1014.559,136.847,-123.440,166.604,56.263,160.305
C08738=1014.555,136.598,-123.421,166.602,56.274,160.307
C08739=1014.551,136.349,-123.403,166.598,56.285,160.308
C08740=1014.547,136.099,-123.385,166.596,56.296,160.310
C08741=1014.542,135.850,-123.367,166.592,56.307,160.311
C08742=1014.538,135.600,-123.348,166.589,56.319,160.313
C08743=1014.534,135.352,-123.330,166.586,56.330,160.314
C08744=1014.529,135.102,-123.312,166.583,56.341,160.316
C08745=1014.525,134.853,-123.293,166.580,56.353,160.317
C08746=1014.520,134.603,-123.275,166.576,56.364,160.319
C08747=1014.517,134.354,-123.256,166.574,56.375,160.320
C08748=1014.512,134.105,-123.238,166.570,56.386,160.322
C08749=1014.507,133.856,-123.220,166.567,56.397,160.323
C08750=1014.503,133.606,-123.201,166.564,56.408,160.325
C08751=1014.499,133.357,-123.184,166.561,56.419,160.326
C08752=1014.495,133.108,-123.165,166.557,56.430,160.327
C08753=1014.490,132.858,-123.147,166.555,56.442,160.329
C08754=1014.486,132.610,-123.129,166.551,56.453,160.330
C08755=1014.482,132.360,-123.110,166.549,56.464,160.332
C08756=1014.477,132.111,-123.092,166.545,56.475,160.333
C08757=1014.472,131.861,-123.074,166.543,56.486,160.335
C08758=1014.469,131.612,-123.055,166.540,56.497,160.337
C08759=1014.464,131.363,-123.037,166.537,56.509,160.338
C08760=1014.460,131.113,-123.019,166.534,56.519,160.340
C08761=1014.456,130.865,-123.001,166.531,56.531,160.341
C08762=1014.451,130.615,-122.983,166.528,56.541,160.343
C08763=1014.447,130.365,-122.965,166.525,56.553,160.344
C08764=1014.443,130.116,-122.947,166.522,56.564,160.346
C08765=1014.439,129.867,-122.928,166.518,56.576,160.347
C08766=1014.434,129.617,-122.910,166.516,56.586,160.349
C08767=1014.430,129.369,-122.892,166.513,56.597,160.350
C08768=1014.426,129.119,-122.875,166.510,56.608,160.351
C08769=1014.421,128.869,-122.856,166.507,56.620,160.353
C08770=1014.417,128.621,-122.839,166.504,56.631,160.354
C08771=1014.413,128.370,-122.821,166.500,56.643,160.356
C08772=1014.408,128.121,-122.802,166.498,56.653,160.357
C08773=1014.404,127.872,-122.785,166.494,56.665,160.359
C08774=1014.400,127.622,-122.767,166.492,56.676,160.361
C08775=1014.395,127.373,-122.749,166.488,56.687,160.362
C08776=1014.391,127.124,-122.731,166.486,56.699,160.364
C08777=1014.386,126.874,-122.714,166.482,56.710,160.365
C08778=1014.382,126.626,-122.696,166.480,56.721,160.367
C08779=1014.378,126.376,-122.679,166.476,56.732,160.368
C08780=1014.373,126.127,-122.660,166.474,56.743,160.370
C08781=1014.369,125.878,-122.643,166.471,56.754,160.371
C08782=1014.364,125.628,-122.625,166.468,56.766,160.373
C08783=1014.360,125.379,-122.607,166.465,56.776,160.374
C08784=1014.355,125.129,-122.590,166.462,56.788,160.376
C08785=1014.351,124.880,-122.572,166.459,56.799,160.377
C08786=1014.347,124.631,-122.555,166.456,56.811,160.379
C08787=1014.342,124.381,-122.536,166.454,56.821,160.380
C08788=1014.338,124.133,-122.519,166.450,56.833,160.382
C08789=1014.333,123.883,-122.501,166.448,56.844,160.383
C08790=1014.329,123.633,-122.483,166.445,56.855,160.385
C08791=1014.325,123.384,-122.466,166.442,56.866,160.386
C08792=1014.320,123.135,-122.448,166.440,56.877,160.388
C08793=1014.316,122.855,-122.428,166.435,56.890,160.389
C08794=1014.310,122.574,-122.409,166.433,56.902,160.391
C08795=1014.305,122.294,-122.389,166.429,56.915,160.393
C08796=1014.301,122.014,-122.369,166.426,56.927,160.395
C08797=1014.296,121.765,-122.351,166.424,56.938,160.396
C08798=1014.292,121.515,-122.334,166.420,56.949,160.398
C08799=1014.288,121.265,-122.316,166.417,56.960,160.399
C08800=1014.284,121.017,-122.298,166.415,56.972,160.401
C08801=1014.279,120.767,-122.281,166.412,56.983,160.402
C08802=1014.275,120.518,-122.263,166.409,56.993,160.403
C08803=1014.271,120.268,-122.246,166.407,57.005,160.405
C08804=1014.267,120.019,-122.228,166.403,57.016,160.407
C08805=1014.262,119.769,-122.210,166.400,57.026,160.408
C08806=1014.258,119.521,-122.193,166.398,57.038,160.410
C08807=1014.253,119.271,-122.175,166.395,57.049,160.411
C08808=1014.249,119.022,-122.157,166.392,57.060,160.413
C08809=1014.245,118.772,-122.140,166.390,57.071,160.414
C08810=1014.241,118.523,-122.123,166.387,57.082,160.416
C08811=1014.236,118.274,-122.105,166.383,57.093,160.417
C08812=1014.232,118.024,-122.088,166.381,57.103,160.418
C08813=1014.227,117.775,-122.069,166.379,57.115,160.420
C08814=1014.224,117.526,-122.052,166.376,57.126,160.422
C08815=1014.219,117.276,-122.035,166.372,57.137,160.423
C08816=1014.215,117.027,-122.017,166.370,57.147,160.424
C08817=1014.210,116.777,-122.000,166.368,57.159,160.426
C08818=1014.206,116.528,-121.982,166.365,57.169,160.428
C08819=1014.202,116.279,-121.965,166.361,57.181,160.429
C08820=1014.198,116.029,-121.947,166.359,57.191,160.431
C08821=1014.194,115.781,-121.930,166.356,57.202,160.432
C08822=1014.189,115.531,-121.912,166.354,57.213,160.434
C08823=1014.185,115.281,-121.895,166.352,57.224,160.435
C08824=1014.181,115.032,-121.877,166.348,57.235,160.437
C08825=1014.177,114.783,-121.860,166.345,57.246,160.438
C08826=1014.173,114.533,-121.843,166.343,57.257,160.439
C08827=1014.168,114.284,-121.825,166.340,57.267,160.441
C08828=1014.164,114.035,-121.807,166.337,57.278,160.442
C08829=1014.160,113.785,-121.790,166.334,57.290,160.444
C08830=1014.156,113.536,-121.772,166.332,57.301,160.446
C08831=1014.152,113.287,-121.755,166.329,57.311,160.447
C08832=1014.147,113.037,-121.738,166.327,57.322,160.449
C08833=1014.143,112.788,-121.721,166.324,57.333,160.450
C08834=1014.139,112.539,-121.703,166.321,57.344,160.451
C08835=1014.135,112.289,-121.685,166.319,57.354,160.453
C08836=1014.131,112.040,-121.668,166.316,57.365,160.454
C08837=1014.126,111.790,-121.650,166.313,57.376,160.456
C08838=1014.122,111.541,-121.633,166.310,57.387,160.457
C08839=1014.118,111.292,-121.617,166.308,57.398,160.459
C08840=1014.113,111.042,-121.599,166.306,57.409,160.461
C08841=1014.109,110.793,-121.582,166.303,57.420,160.462
C08842=1014.105,110.544,-121.565,166.299,57.431,160.463
C08843=1014.100,110.294,-121.548,166.297,57.442,160.465
C08844=1014.096,110.045,-121.531,166.294,57.452,160.466
C08845=1014.092,109.795,-121.514,166.292,57.463,160.468
C08846=1014.087,109.546,-121.497,166.290,57.475,160.470
C08847=1014.083,109.297,-121.480,166.287,57.485,160.471
C08848=1014.079,109.047,-121.463,166.284,57.497,160.472
C08849=1014.074,108.798,-121.446,166.281,57.507,160.474
C08850=1014.070,108.548,-121.429,166.279,57.518,160.475
C08851=1014.066,108.299,-121.413,166.276,57.529,160.477
C08852=1014.061,108.049,-121.395,166.274,57.540,160.479
C08853=1014.057,107.800,-121.379,166.271,57.552,160.480
C08854=1014.053,107.551,-121.362,166.268,57.562,160.482
C08855=1014.048,107.302,-121.345,166.265,57.573,160.483
C08856=1014.044,107.052,-121.328,166.263,57.584,160.485
C08857=1014.039,106.772,-121.309,166.261,57.596,160.486
C08858=1014.034,106.491,-121.290,166.257,57.609,160.488
C08859=1014.029,106.211,-121.271,166.254,57.621,160.489
C08860=1014.024,105.932,-121.252,166.251,57.633,160.491
C08861=1014.020,105.683,-121.235,166.249,57.644,160.493
C08862=1014.015,105.432,-121.219,166.246,57.655,160.494
C08863=1014.011,105.183,-121.202,166.244,57.666,160.496
C08864=1014.007,104.934,-121.185,166.241,57.677,160.497
C08865=1014.003,104.685,-121.168,166.239,57.687,160.499
C08866=1013.998,104.435,-121.151,166.235,57.699,160.500
C08867=1013.994,104.186,-121.134,166.233,57.709,160.502
C08868=1013.989,103.937,-121.118,166.230,57.720,160.503
C08869=1013.985,103.687,-121.102,166.228,57.731,160.505
C08870=1013.980,103.437,-121.085,166.225,57.742,160.506
C08871=1013.976,103.188,-121.068,166.223,57.752,160.508
C08872=1013.972,102.939,-121.051,166.220,57.763,160.509
C08873=1013.968,102.690,-121.034,166.218,57.774,160.511
C08874=1013.963,102.440,-121.018,166.216,57.785,160.512
C08875=1013.959,102.190,-121.001,166.213,57.796,160.514
C08876=1013.954,101.941,-120.984,166.211,57.806,160.515
C08877=1013.951,101.692,-120.967,166.208,57.817,160.517
C08878=1013.945,101.442,-120.950,166.206,57.828,160.518
C08879=1013.942,101.193,-120.934,166.203,57.838,160.520
C08880=1013.937,100.944,-120.918,166.200,57.849,160.521
C08881=1013.933,100.694,-120.900,166.198,57.860,160.523
C08882=1013.929,100.445,-120.884,166.195,57.871,160.524
C08883=1013.925,100.195,-120.867,166.193,57.881,160.526
C08884=1013.921,99.945,-120.850,166.190,57.892,160.527
C08885=1013.916,99.697,-120.834,166.188,57.903,160.529
C08886=1013.912,99.447,-120.817,166.185,57.913,160.530
C08887=1013.908,99.198,-120.801,166.183,57.924,160.532
C08888=1013.904,98.948,-120.784,166.180,57.935,160.533
C08889=1013.899,98.699,-120.767,166.178,57.946,160.535
C08890=1013.895,98.449,-120.751,166.175,57.956,160.536
C08891=1013.890,98.200,-120.735,166.173,57.967,160.538
C08892=1013.886,97.950,-120.718,166.171,57.978,160.539
C08893=1013.882,97.701,-120.702,166.168,57.989,160.541
C08894=1013.877,97.452,-120.685,166.166,58.000,160.542
C08895=1013.872,97.202,-120.669,166.163,58.010,160.544
C08896=1013.868,96.953,-120.653,166.160,58.021,160.545
C08897=1013.864,96.703,-120.636,166.158,58.031,160.547
C08898=1013.859,96.454,-120.620,166.156,58.042,160.548
C08899=1013.855,96.205,-120.604,166.153,58.053,160.550
C08900=1013.850,95.956,-120.588,166.151,58.064,160.551
C08901=1013.846,95.705,-120.571,166.148,58.075,160.553
C08902=1013.842,95.456,-120.554,166.146,58.086,160.554
C08903=1013.837,95.207,-120.539,166.143,58.096,160.556
C08904=1013.833,94.958,-120.522,166.141,58.107,160.557
C08905=1013.828,94.708,-120.506,166.138,58.117,160.559
C08906=1013.825,94.459,-120.489,166.136,58.128,160.560
C08907=1013.820,94.209,-120.474,166.134,58.139,160.562
C08908=1013.816,93.960,-120.458,166.131,58.149,160.563
C08909=1013.811,93.710,-120.441,166.128,58.160,160.564
C08910=1013.806,93.460,-120.425,166.126,58.171,160.566
C08911=1013.803,93.211,-120.408,166.123,58.181,160.567
C08912=1013.798,92.962,-120.392,166.122,58.191,160.569
C08913=1013.794,92.713,-120.376,166.119,58.202,160.571
C08914=1013.789,92.463,-120.360,166.117,58.213,160.572
C08915=1013.785,92.214,-120.344,166.114,58.223,160.573
C08916=1013.781,91.964,-120.327,166.112,58.234,160.575
C08917=1013.777,91.715,-120.311,166.110,58.245,160.576
C08918=1013.772,91.466,-120.295,166.107,58.255,160.578
C08919=1013.768,91.216,-120.279,166.105,58.266,160.579
C08920=1013.763,90.967,-120.263,166.103,58.276,160.581
C08921=1013.759,90.687,-120.244,166.100,58.288,160.582
C08922=1013.754,90.406,-120.226,166.097,58.300,160.584
C08923=1013.749,90.127,-120.208,166.094,58.312,160.586
C08924=1013.745,89.847,-120.190,166.092,58.324,160.588
C08925=1013.740,89.598,-120.174,166.090,58.334,160.589
C08926=1013.736,89.349,-120.158,166.087,58.345,160.590
C08927=1013.731,89.099,-120.142,166.084,58.355,160.592
C08928=1013.728,88.850,-120.125,166.083,58.365,160.593
C08929=1013.723,88.600,-120.109,166.080,58.375,160.595
C08930=1013.719,88.351,-120.093,166.078,58.386,160.596
C08931=1013.714,88.100,-120.077,166.076,58.397,160.598
C08932=1013.709,87.852,-120.061,166.073,58.407,160.599
C08933=1013.704,87.602,-120.046,166.070,58.418,160.601
C08934=1013.700,87.353,-120.030,166.069,58.429,160.602
C08935=1013.696,87.103,-120.014,166.066,58.439,160.604
C08936=1013.691,86.853,-119.998,166.064,58.450,160.605
C08937=1013.687,86.604,-119.982,166.061,58.460,160.606
C08938=1013.683,86.354,-119.967,166.059,58.471,160.608
C08939=1013.678,86.105,-119.950,166.057,58.482,160.610
C08940=1013.674,85.856,-119.934,166.055,58.491,160.611
C08941=1013.669,85.606,-119.919,166.053,58.502,160.613
C08942=1013.665,85.357,-119.904,166.050,58.512,160.614
C08943=1013.660,85.107,-119.888,166.047,58.523,160.615
C08944=1013.656,84.858,-119.872,166.045,58.534,160.617
C08945=1013.652,84.608,-119.856,166.043,58.544,160.618
C08946=1013.647,84.359,-119.840,166.041,58.554,160.620
